KUKA KRL program: EPS_2_251497_STMH_A_20251003030554.src

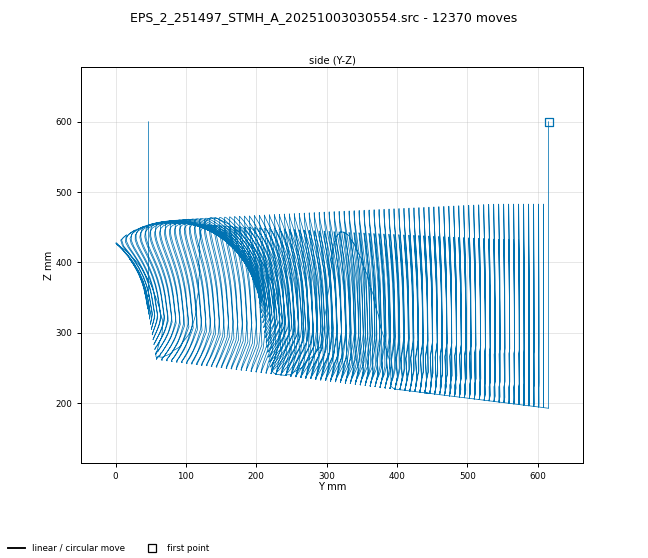
[picture p0: tool path of EPS_2_251497_STMH_A_20251003030554.src, 12370 of 12372 moves have a stored position in this frame; points joined in program order, loops and branches not executed]
&ACCESS RVP
&REL 4
&COMMENT QRS 19112012
&PARAM EDITMASK = *
DEF PART()
EXT BAS (BAS_COMMAND :IN,REAL :IN )
INT I
BAS (#INITMOV,0 )

;KUKA QRS Post kuka4.cps  Date:22-06-2017 !

File_ID=2874

QRS_PRE_INIT()

;Init var - Until changes are made in qrs_pre_init
Outlet_Square_prg=0
Inlet_1_Square_prg=0
Inlet_2_Square_prg=0
Inlet_3_Square_prg=0
Inlet_4_Square_prg=0
Inlet_5_Square_prg=0

Outlet_1={X 0.000, Y 540.910, Z 382.500, B 0.000, E1 0.000 }
Inlet_1={X 0.000, Y 544.470, Z 332.500, B 0.000, E1 230.000 }
Outlet_1_type=201
Inlet_1_type=201
;QRS#1=Sidecore dimensions
;QRS#2=200-8" PVC SDR 35
;QRS#3=200-8" PVC SDR 35
;QRS#4=
;QRS#5=
;QRS#6=
;QRS#7=
;QRS#8=
;QRS#9=12-08 PSX
;QRS#10=12-08 PSX
;QRS#11=
;QRS#12=
;QRS#13=
;QRS#14=
;QRS#15=
;QRS#16=1220x127x762 2,5'
;QRS#17=EPS Height
;QRS#18=483
;QRS#19=*
;QRS#20= UPDATED VERSION 22-06-2017
;QRS#21=*
Outlet_Square=0100
Inlet_1_Square=0100
Inlet_2_Square=0
Inlet_3_Square=0
Inlet_4_Square=0
Inlet_5_Square=0
Mill_Square=1
Outlet_Square_Prg=204
Inlet_1_Square_prg=204

QRS_INIT()

$ADVANCE=5

; T1
PTP {E1 173.565,E2 173.565}
PTP {X 0,Y 615.49,A -85,B 0,C 180,E1 173.565,E2 173.565,E3 0,E4 0,E5 0,E6 0}
QRS_SPEED_INIT()
LIN {X 0,Y 615.49,Z 600,A -85,B 0,C 180,E1 173.565,E2 173.565,E3 0,E4 0,E5 0,E6 0} C_VEL
LIN {X 0,Y 615.49,Z 202.871,A -85,B 0,C 180,E1 173.565,E2 173.565} C_VEL
LIN {X 0,Y 615.49,Z 194.7,A -85,B 0,C 180,E1 173.565,E2 173.565} C_VEL
LIN {X 0,Y 615.472,Z 192.7,A -85,B 0,C 180,E1 173.379,E2 173.379} C_VEL
LIN {X 0,Y 615.458,Z 192.696,A -85,B 0,C 180,E1 170.801,E2 170.801} C_VEL
LIN {X 0,Y 615.425,Z 192.697,A -85,B 0,C 180,E1 168.138,E2 168.138} C_VEL
LIN {X 0,Y 615.478,Z 192.701,A -85,B 0,C 180,E1 165.451,E2 165.451} C_VEL
LIN {X 0,Y 615.445,Z 192.694,A -85,B 0,C 180,E1 162.729,E2 162.729} C_VEL
LIN {X 0,Y 615.439,Z 192.695,A -85,B 0,C 180,E1 160.661,E2 160.661} C_VEL
LIN {X 0,Y 615.434,Z 192.695,A -85,B 0,C 180,E1 158.566,E2 158.566} C_VEL
LIN {X 0,Y 615.447,Z 192.698,A -85,B 0,C 180,E1 155.986,E2 155.986} C_VEL
LIN {X 0,Y 615.494,Z 192.701,A -85,B 0,C 180,E1 153.556,E2 153.556} C_VEL
LIN {X 0,Y 615.489,Z 192.693,A -85,B 0,C 180,E1 151.342,E2 151.342} C_VEL
LIN {X 0,Y 615.451,Z 192.692,A -85,B 0,C 180,E1 148.909,E2 148.909} C_VEL
LIN {X 0,Y 615.438,Z 192.695,A -85,B 0,C 180,E1 146.463,E2 146.463} C_VEL
LIN {X 0,Y 615.454,Z 192.697,A -85,B 0,C 180,E1 144.162,E2 144.162} C_VEL
LIN {X 0,Y 615.483,Z 192.699,A -85,B 0,C 180,E1 141.931,E2 141.931} C_VEL
LIN {X 0,Y 615.489,Z 192.688,A -85,B 0,C 180,E1 139.394,E2 139.394} C_VEL
LIN {X 0,Y 615.441,Z 192.694,A -85,B 0,C 180,E1 136.752,E2 136.752} C_VEL
LIN {X 0,Y 615.483,Z 192.702,A -85,B 0,C 180,E1 133.997,E2 133.997} C_VEL
LIN {X 0,Y 615.456,Z 192.69,A -85,B 0,C 180,E1 131.091,E2 131.091} C_VEL
LIN {X 0,Y 615.446,Z 192.692,A -85,B 0,C 180,E1 128.902,E2 128.902} C_VEL
LIN {X 0,Y 615.466,Z 192.697,A -85,B 0,C 180,E1 126.421,E2 126.421} C_VEL
LIN {X 0,Y 615.487,Z 192.686,A -85,B 0,C 180,E1 123.535,E2 123.535} C_VEL
LIN {X 0,Y 615.452,Z 192.692,A -85,B 0,C 180,E1 120.918,E2 120.918} C_VEL
LIN {X 0,Y 615.473,Z 192.699,A -85,B 0,C 180,E1 118.448,E2 118.448} C_VEL
LIN {X 0,Y 615.483,Z 192.685,A -85,B 0,C 180,E1 115.568,E2 115.568} C_VEL
LIN {X 0,Y 615.461,Z 192.694,A -85,B 0,C 180,E1 112.843,E2 112.843} C_VEL
LIN {X 0,Y 615.491,Z 192.69,A -85,B 0,C 180,E1 110.03,E2 110.03} C_VEL
LIN {X 0,Y 615.461,Z 192.689,A -85,B 0,C 180,E1 107.269,E2 107.269} C_VEL
LIN {X 0,Y 615.488,Z 192.702,A -85,B 0,C 180,E1 104.547,E2 104.547} C_VEL
LIN {X 0,Y 615.486,Z 192.685,A -85,B 0,C 180,E1 101.859,E2 101.859} C_VEL
LIN {X 0,Y 615.462,Z 192.692,A -85,B 0,C 180,E1 99.198,E2 99.198} C_VEL
LIN {X 0,Y 615.489,Z 192.698,A -85,B 0,C 180,E1 96.556,E2 96.556} C_VEL
LIN {X 0,Y 615.486,Z 192.684,A -85,B 0,C 180,E1 93.928,E2 93.928} C_VEL
LIN {X 0,Y 615.464,Z 192.692,A -85,B 0,C 180,E1 91.308,E2 91.308} C_VEL
LIN {X 0,Y 615.489,Z 192.698,A -85,B 0,C 180,E1 88.692,E2 88.692} C_VEL
LIN {X 0,Y 615.487,Z 192.683,A -85,B 0,C 180,E1 86.072,E2 86.072} C_VEL
LIN {X 0,Y 615.468,Z 192.692,A -85,B 0,C 180,E1 83.436,E2 83.436} C_VEL
LIN {X 0,Y 615.487,Z 192.697,A -85,B 0,C 180,E1 80.802,E2 80.802} C_VEL
LIN {X 0,Y 615.487,Z 192.683,A -85,B 0,C 180,E1 78.14,E2 78.14} C_VEL
LIN {X 0,Y 615.476,Z 192.693,A -85,B 0,C 180,E1 75.452,E2 75.452} C_VEL
LIN {X 0,Y 615.481,Z 192.692,A -85,B 0,C 180,E1 72.731,E2 72.731} C_VEL
LIN {X 0,Y 615.482,Z 192.685,A -85,B 0,C 180,E1 69.969,E2 69.969} C_VEL
LIN {X 0,Y 615.49,Z 192.7,A -85,B 0,C 180,E1 67.158,E2 67.158} C_VEL
LIN {X 0,Y 615.499,Z 192.68,A -85,B 0,C 180,E1 64.288,E2 64.288} C_VEL
LIN {X 0,Y 615.486,Z 192.703,A -85,B 0,C 180,E1 61.345,E2 61.345} C_VEL
LIN {X 0,Y 615.476,Z 192.691,A -85,B 0,C 180,E1 58.915,E2 58.915} C_VEL
LIN {X 0,Y 615.48,Z 192.89,A -85,B 0,C 180,E1 57.954,E2 57.954} C_VEL
LIN {X 0,Y 615.463,Z 208.033,A -85,B 0,C 180,E1 55.302,E2 55.302} C_VEL
LIN {X 0,Y 615.454,Z 222.372,A -85,B 0,C 180,E1 52.818,E2 52.818} C_VEL
LIN {X 0,Y 615.432,Z 329.039,A -85,B 0,C 180,E1 51.542,E2 51.542} C_VEL
LIN {X 0,Y 615.439,Z 342.064,A -85,B 0,C 180,E1 51.255,E2 51.255} C_VEL
LIN {X 0,Y 615.473,Z 354.262,A -85,B 0,C 180,E1 50.856,E2 50.856} C_VEL
LIN {X 0,Y 615.491,Z 365.958,A -85,B 0,C 180,E1 50.342,E2 50.342} C_VEL
LIN {X 0,Y 615.479,Z 377.926,A -85,B 0,C 180,E1 49.656,E2 49.656} C_VEL
LIN {X 0,Y 615.496,Z 388.354,A -85,B 0,C 180,E1 48.904,E2 48.904} C_VEL
LIN {X 0,Y 615.499,Z 397.717,A -85,B 0,C 180,E1 48.073,E2 48.073} C_VEL
LIN {X 0,Y 615.496,Z 406.315,A -85,B 0,C 180,E1 47.128,E2 47.128} C_VEL
LIN {X 0,Y 615.495,Z 413.248,A -85,B 0,C 180,E1 46.192,E2 46.192} C_VEL
LIN {X 0,Y 615.496,Z 419.897,A -85,B 0,C 180,E1 45.067,E2 45.067} C_VEL
LIN {X 0,Y 615.493,Z 424.69,A -85,B 0,C 180,E1 44.005,E2 44.005} C_VEL
LIN {X 0,Y 615.495,Z 427.941,A -85,B 0,C 180,E1 43.055,E2 43.055} C_VEL
LIN {X 0,Y 615.496,Z 430.296,A -85,B 0,C 180,E1 42.088,E2 42.088} C_VEL
LIN {X 0,Y 615.494,Z 431.771,A -85,B 0,C 180,E1 41.102,E2 41.102} C_VEL
LIN {X 0,Y 615.492,Z 432.346,A -85,B 0,C 180,E1 39.749,E2 39.749} C_VEL
LIN {X 0,Y 615.494,Z 431.883,A -85,B 0,C 180,E1 38.904,E2 38.904} C_VEL
LIN {X 0,Y 615.494,Z 430.657,A -85,B 0,C 180,E1 38.021,E2 38.021} C_VEL
LIN {X 0,Y 615.497,Z 428.187,A -85,B 0,C 180,E1 36.946,E2 36.946} C_VEL
LIN {X 0,Y 615.496,Z 424.457,A -85,B 0,C 180,E1 35.844,E2 35.844} C_VEL
LIN {X 0,Y 615.495,Z 419.188,A -85,B 0,C 180,E1 34.711,E2 34.711} C_VEL
LIN {X 0,Y 615.496,Z 412.08,A -85,B 0,C 180,E1 33.545,E2 33.545} C_VEL
LIN {X 0,Y 615.499,Z 405.237,A -85,B 0,C 180,E1 32.651,E2 32.651} C_VEL
LIN {X 0,Y 615.497,Z 397.831,A -85,B 0,C 180,E1 31.849,E2 31.849} C_VEL
LIN {X 0,Y 615.496,Z 388.386,A -85,B 0,C 180,E1 31.008,E2 31.008} C_VEL
LIN {X 0,Y 615.472,Z 377.947,A -85,B 0,C 180,E1 30.255,E2 30.255} C_VEL
LIN {X 0,Y 615.467,Z 366.665,A -85,B 0,C 180,E1 29.604,E2 29.604} C_VEL
LIN {X 0,Y 615.495,Z 354.87,A -85,B 0,C 180,E1 29.078,E2 29.078} C_VEL
LIN {X 0,Y 615.488,Z 342.102,A -85,B 0,C 180,E1 28.658,E2 28.658} C_VEL
LIN {X 0,Y 615.477,Z 330.305,A -85,B 0,C 180,E1 28.392,E2 28.392} C_VEL
LIN {X 0,Y 615.472,Z 295.985,A -85,B 0,C 180,E1 27.967,E2 27.967} C_VEL
LIN {X 0,Y 615.484,Z 222.337,A -85,B 0,C 180,E1 27.087,E2 27.087} C_VEL
LIN {X 0,Y 615.491,Z 206.092,A -85,B 0,C 180,E1 24.272,E2 24.272} C_VEL
LIN {X 0,Y 615.439,Z 192.697,A -85,B 0,C 180,E1 21.917,E2 21.917} C_VEL
LIN {X 0,Y 615.443,Z 192.698,A -85,B 0,C 180,E1 20.034,E2 20.034} C_VEL
LIN {X 0,Y 615.435,Z 192.697,A -85,B 0,C 180,E1 17.958,E2 17.958} C_VEL
LIN {X 0,Y 615.431,Z 192.697,A -85,B 0,C 180,E1 15.906,E2 15.906} C_VEL
LIN {X 0,Y 615.428,Z 192.697,A -85,B 0,C 180,E1 13.875,E2 13.875} C_VEL
LIN {X 0,Y 615.425,Z 192.697,A -85,B 0,C 180,E1 11.862,E2 11.862} C_VEL
LIN {X 0,Y 615.458,Z 192.695,A -85,B 0,C 180,E1 9.199,E2 9.199} C_VEL
LIN {X 0,Y 615.464,Z 192.7,A -85,B 0,C 180,E1 6.557,E2 6.557} C_VEL
LIN {X 0,Y 615.42,Z 192.698,A -85,B 0,C 180,E1 3.929,E2 3.929} C_VEL
LIN {X 0,Y 615.454,Z 192.697,A -85,B 0,C 180,E1 1.308,E2 1.308} C_VEL
LIN {X 0,Y 615.461,Z 192.7,A -85,B 0,C 180,E1 -1.309,E2 -1.309} C_VEL
LIN {X 0,Y 615.414,Z 192.699,A -85,B 0,C 180,E1 -3.929,E2 -3.929} C_VEL
LIN {X 0,Y 615.452,Z 192.699,A -85,B 0,C 180,E1 -6.604,E2 -6.604} C_VEL
LIN {X 0,Y 615.455,Z 192.7,A -85,B 0,C 180,E1 -9.2,E2 -9.2} C_VEL
LIN {X 0,Y 615.412,Z 192.7,A -85,B 0,C 180,E1 -11.863,E2 -11.863} C_VEL
LIN {X 0,Y 615.462,Z 192.7,A -85,B 0,C 180,E1 -14.55,E2 -14.55} C_VEL
LIN {X 0,Y 615.439,Z 192.698,A -85,B 0,C 180,E1 -17.272,E2 -17.272} C_VEL
LIN {X 0,Y 615.432,Z 192.698,A -85,B 0,C 180,E1 -19.34,E2 -19.34} C_VEL
LIN {X 0,Y 615.426,Z 192.698,A -85,B 0,C 180,E1 -21.434,E2 -21.434} C_VEL
LIN {X 0,Y 615.421,Z 192.698,A -85,B 0,C 180,E1 -23.559,E2 -23.559} C_VEL
LIN {X 0,Y 615.421,Z 192.698,A -85,B 0,C 180,E1 -25.719,E2 -25.719} C_VEL
LIN {X 0,Y 615.484,Z 192.701,A -85,B 0,C 180,E1 -28.461,E2 -28.461} C_VEL
LIN {X 0,Y 615.446,Z 192.695,A -85,B 0,C 180,E1 -31.09,E2 -31.09} C_VEL
LIN {X 0,Y 615.431,Z 192.696,A -85,B 0,C 180,E1 -33.24,E2 -33.24} C_VEL
LIN {X 0,Y 615.428,Z 192.697,A -85,B 0,C 180,E1 -35.62,E2 -35.62} C_VEL
LIN {X 0,Y 615.464,Z 192.699,A -85,B 0,C 180,E1 -38.071,E2 -38.071} C_VEL
LIN {X 0,Y 615.488,Z 192.692,A -85,B 0,C 180,E1 -40.607,E2 -40.607} C_VEL
LIN {X 0,Y 615.434,Z 192.695,A -85,B 0,C 180,E1 -43.25,E2 -43.25} C_VEL
LIN {X 0,Y 615.47,Z 192.7,A -85,B 0,C 180,E1 -46.005,E2 -46.005} C_VEL
LIN {X 0,Y 615.45,Z 192.692,A -85,B 0,C 180,E1 -48.91,E2 -48.91} C_VEL
LIN {X 0,Y 615.438,Z 192.694,A -85,B 0,C 180,E1 -51.097,E2 -51.097} C_VEL
LIN {X 0,Y 615.451,Z 192.697,A -85,B 0,C 180,E1 -53.577,E2 -53.577} C_VEL
LIN {X 0,Y 615.486,Z 192.688,A -85,B 0,C 180,E1 -56.467,E2 -56.467} C_VEL
LIN {X 0,Y 615.443,Z 192.693,A -85,B 0,C 180,E1 -59.082,E2 -59.082} C_VEL
LIN {X 0,Y 615.463,Z 192.697,A -85,B 0,C 180,E1 -61.554,E2 -61.554} C_VEL
LIN {X 0,Y 615.481,Z 192.687,A -85,B 0,C 180,E1 -64.433,E2 -64.433} C_VEL
LIN {X 0,Y 615.447,Z 192.693,A -85,B 0,C 180,E1 -67.046,E2 -67.046} C_VEL
LIN {X 0,Y 615.483,Z 210.777,A -85,B 0,C 180,E1 -69.445,E2 -69.445} C_VEL
LIN {X 0,Y 615.489,Z 232.032,A -85,B 0,C 180,E1 -72.217,E2 -72.217} C_VEL
LIN {X 0,Y 615.494,Z 253.252,A -85,B 0,C 180,E1 -74.945,E2 -74.945} C_VEL
LIN {X 0,Y 615.452,Z 270.312,A -85,B 0,C 180,E1 -77.114,E2 -77.114} C_VEL
LIN {X 0,Y 615.478,Z 378.901,A -85,B 0,C 180,E1 -78.412,E2 -78.412} C_VEL
LIN {X 0,Y 615.47,Z 391.391,A -85,B 0,C 180,E1 -78.683,E2 -78.683} C_VEL
LIN {X 0,Y 615.486,Z 404.642,A -85,B 0,C 180,E1 -79.114,E2 -79.114} C_VEL
LIN {X 0,Y 615.483,Z 416.499,A -85,B 0,C 180,E1 -79.64,E2 -79.64} C_VEL
LIN {X 0,Y 615.495,Z 428.01,A -85,B 0,C 180,E1 -80.305,E2 -80.305} C_VEL
LIN {X 0,Y 615.499,Z 438.353,A -85,B 0,C 180,E1 -81.051,E2 -81.051} C_VEL
LIN {X 0,Y 615.497,Z 446.821,A -85,B 0,C 180,E1 -81.795,E2 -81.795} C_VEL
LIN {X 0,Y 615.496,Z 455.971,A -85,B 0,C 180,E1 -82.785,E2 -82.785} C_VEL
LIN {X 0,Y 615.497,Z 463.319,A -85,B 0,C 180,E1 -83.773,E2 -83.773} C_VEL
LIN {X 0,Y 615.498,Z 469.207,A -85,B 0,C 180,E1 -84.759,E2 -84.759} C_VEL
LIN {X 0,Y 615.494,Z 473.853,A -85,B 0,C 180,E1 -85.744,E2 -85.744} C_VEL
LIN {X 0,Y 615.494,Z 477.4,A -85,B 0,C 180,E1 -86.727,E2 -86.727} C_VEL
LIN {X 0,Y 615.497,Z 479.233,A -85,B 0,C 180,E1 -87.382,E2 -87.382} C_VEL
LIN {X 0,Y 615.499,Z 480.608,A -85,B 0,C 180,E1 -88.037,E2 -88.037} C_VEL
LIN {X 0,Y 615.496,Z 482.173,A -85,B 0,C 180,E1 -89.346,E2 -89.346} C_VEL
LIN {X 0,Y 615.494,Z 482.389,A -85,B 0,C 180,E1 -90,E2 -90} C_VEL
LIN {X 0,Y 615.495,Z 481.58,A -85,B 0,C 180,E1 -91.308,E2 -91.308} C_VEL
LIN {X 0,Y 615.499,Z 480.608,A -85,B 0,C 180,E1 -91.963,E2 -91.963} C_VEL
LIN {X 0,Y 615.497,Z 479.234,A -85,B 0,C 180,E1 -92.617,E2 -92.617} C_VEL
LIN {X 0,Y 615.496,Z 476.351,A -85,B 0,C 180,E1 -93.6,E2 -93.6} C_VEL
LIN {X 0,Y 615.498,Z 472.444,A -85,B 0,C 180,E1 -94.584,E2 -94.584} C_VEL
LIN {X 0,Y 615.499,Z 467.409,A -85,B 0,C 180,E1 -95.569,E2 -95.569} C_VEL
LIN {X 0,Y 615.496,Z 460.87,A -85,B 0,C 180,E1 -96.583,E2 -96.583} C_VEL
LIN {X 0,Y 615.497,Z 453.141,A -85,B 0,C 180,E1 -97.544,E2 -97.544} C_VEL
LIN {X 0,Y 615.498,Z 445.056,A -85,B 0,C 180,E1 -98.37,E2 -98.37} C_VEL
LIN {X 0,Y 615.499,Z 435.182,A -85,B 0,C 180,E1 -99.198,E2 -99.198} C_VEL
LIN {X 0,Y 615.492,Z 424.001,A -85,B 0,C 180,E1 -99.944,E2 -99.944} C_VEL
LIN {X 0,Y 615.485,Z 413.049,A -85,B 0,C 180,E1 -100.526,E2 -100.526} C_VEL
LIN {X 0,Y 615.476,Z 400.523,A -85,B 0,C 180,E1 -101.039,E2 -101.039} C_VEL
LIN {X 0,Y 615.471,Z 388.127,A -85,B 0,C 180,E1 -101.401,E2 -101.401} C_VEL
LIN {X 0,Y 615.482,Z 374.566,A -85,B 0,C 180,E1 -101.651,E2 -101.651} C_VEL
LIN {X 0,Y 615.452,Z 270.313,A -85,B 0,C 180,E1 -102.886,E2 -102.886} C_VEL
LIN {X 0,Y 615.487,Z 249.274,A -85,B 0,C 180,E1 -105.563,E2 -105.563} C_VEL
LIN {X 0,Y 615.456,Z 227.017,A -85,B 0,C 180,E1 -108.434,E2 -108.434} C_VEL
LIN {X 0,Y 615.482,Z 206.801,A -85,B 0,C 180,E1 -111.079,E2 -111.079} C_VEL
LIN {X 0,Y 615.447,Z 192.693,A -85,B 0,C 180,E1 -112.977,E2 -112.977} C_VEL
LIN {X 0,Y 615.499,Z 192.686,A -85,B 0,C 180,E1 -115.712,E2 -115.712} C_VEL
LIN {X 0,Y 615.449,Z 192.695,A -85,B 0,C 180,E1 -118.656,E2 -118.656} C_VEL
LIN {X 0,Y 615.447,Z 192.692,A -85,B 0,C 180,E1 -121.079,E2 -121.079} C_VEL
LIN {X 0,Y 615.493,Z 192.701,A -85,B 0,C 180,E1 -124.017,E2 -124.017} C_VEL
LIN {X 0,Y 615.451,Z 192.697,A -85,B 0,C 180,E1 -126.422,E2 -126.422} C_VEL
LIN {X 0,Y 615.444,Z 192.693,A -85,B 0,C 180,E1 -129.057,E2 -129.057} C_VEL
LIN {X 0,Y 615.487,Z 192.69,A -85,B 0,C 180,E1 -131.468,E2 -131.468} C_VEL
LIN {X 0,Y 615.459,Z 192.698,A -85,B 0,C 180,E1 -134.146,E2 -134.146} C_VEL
LIN {X 0,Y 615.435,Z 192.695,A -85,B 0,C 180,E1 -136.75,E2 -136.75} C_VEL
LIN {X 0,Y 615.488,Z 192.692,A -85,B 0,C 180,E1 -139.393,E2 -139.393} C_VEL
LIN {X 0,Y 615.458,Z 192.699,A -85,B 0,C 180,E1 -141.983,E2 -141.983} C_VEL
LIN {X 0,Y 615.428,Z 192.697,A -85,B 0,C 180,E1 -144.38,E2 -144.38} C_VEL
LIN {X 0,Y 615.433,Z 192.696,A -85,B 0,C 180,E1 -146.76,E2 -146.76} C_VEL
LIN {X 0,Y 615.463,Z 192.694,A -85,B 0,C 180,E1 -149.079,E2 -149.079} C_VEL
LIN {X 0,Y 615.485,Z 192.701,A -85,B 0,C 180,E1 -151.538,E2 -151.538} C_VEL
LIN {X 0,Y 615.422,Z 192.698,A -85,B 0,C 180,E1 -154.281,E2 -154.281} C_VEL
LIN {X 0,Y 615.484,Z 192.696,A -85,B 0,C 180,E1 -157.155,E2 -157.155} C_VEL
LIN {X 0,Y 615.426,Z 192.699,A -85,B 0,C 180,E1 -159.965,E2 -159.965} C_VEL
LIN {X 0,Y 615.42,Z 192.699,A -85,B 0,C 180,E1 -162.041,E2 -162.041} C_VEL
LIN {X 0,Y 615.416,Z 192.699,A -85,B 0,C 180,E1 -164.093,E2 -164.093} C_VEL
LIN {X 0,Y 615.414,Z 192.699,A -85,B 0,C 180,E1 -166.124,E2 -166.124} C_VEL
LIN {X 0,Y 615.453,Z 192.699,A -85,B 0,C 180,E1 -168.806,E2 -168.806} C_VEL
LIN {X 0,Y 615.447,Z 192.7,A -85,B 0,C 180,E1 -171.463,E2 -171.463} C_VEL
LIN {X 0,Y 615.412,Z 192.7,A -85,B 0,C 180,E1 -174.1,E2 -174.1} C_VEL
LIN {X 0,Y 615.46,Z 192.7,A -85,B 0,C 180,E1 -176.727,E2 -176.727} C_VEL
LIN {X 0,Y 615.452,Z 192.698,A -85,B 0,C 180,E1 -179.345,E2 -179.345} C_VEL
LIN {X 0,Y 615.417,Z 192.699,A -85,B 0,C 180,E1 -181.963,E2 -181.963} C_VEL
LIN {X 0,Y 615.462,Z 192.7,A -85,B 0,C 180,E1 -184.585,E2 -184.585} C_VEL
LIN {X 0,Y 615.472,Z 192.7,A -85,B 0,C 180,E1 -186.621,E2 -186.621} C_VEL
LIN {X 0,Y 614.789,Z 192.842,A -85,B 0,C 180,E1 -187.167,E2 -187.167} C_VEL
LIN {X 0,Y 611.948,Z 193.253,A -85,B 0,C 180,E1 -188.053,E2 -188.053} C_VEL
LIN {X 0,Y 609.551,Z 193.564,A -85,B 0,C 180,E1 -188.766,E2 -188.766} C_VEL
LIN {X 0,Y 608.508,Z 193.683,A -85,B 0,C 180,E1 -189.315,E2 -189.315} C_VEL
LIN {X 0,Y 608.415,Z 193.693,A -85,B 0,C 180,E1 -189.501,E2 -189.501} C_VEL
LIN {X 0,Y 608.41,Z 193.694,A -85,B 0,C 180,E1 -192.001,E2 -192.001} C_VEL
LIN {X 0,Y 608.452,Z 193.697,A -85,B 0,C 180,E1 -194.721,E2 -194.721} C_VEL
LIN {X 0,Y 608.448,Z 193.695,A -85,B 0,C 180,E1 -196.784,E2 -196.784} C_VEL
LIN {X 0,Y 608.448,Z 193.693,A -85,B 0,C 180,E1 -198.87,E2 -198.87} C_VEL
LIN {X 0,Y 608.448,Z 193.691,A -85,B 0,C 180,E1 -200.982,E2 -200.982} C_VEL
LIN {X 0,Y 608.424,Z 193.692,A -85,B 0,C 180,E1 -203.125,E2 -203.125} C_VEL
LIN {X 0,Y 608.418,Z 193.693,A -85,B 0,C 180,E1 -205.724,E2 -205.724} C_VEL
LIN {X 0,Y 608.471,Z 193.691,A -85,B 0,C 180,E1 -208.631,E2 -208.631} C_VEL
LIN {X 0,Y 608.431,Z 193.69,A -85,B 0,C 180,E1 -211.318,E2 -211.318} C_VEL
LIN {X 0,Y 608.433,Z 193.692,A -85,B 0,C 180,E1 -213.739,E2 -213.739} C_VEL
LIN {X 0,Y 608.444,Z 193.697,A -85,B 0,C 180,E1 -216.092,E2 -216.092} C_VEL
LIN {X 0,Y 608.447,Z 193.692,A -85,B 0,C 180,E1 -218.589,E2 -218.589} C_VEL
LIN {X 0,Y 608.414,Z 193.692,A -85,B 0,C 180,E1 -221.18,E2 -221.18} C_VEL
LIN {X 0,Y 608.459,Z 193.693,A -85,B 0,C 180,E1 -223.87,E2 -223.87} C_VEL
LIN {X 0,Y 608.455,Z 193.688,A -85,B 0,C 180,E1 -226.692,E2 -226.692} C_VEL
LIN {X 0,Y 608.432,Z 193.69,A -85,B 0,C 180,E1 -228.827,E2 -228.827} C_VEL
LIN {X 0,Y 608.442,Z 193.691,A -85,B 0,C 180,E1 -231.415,E2 -231.415} C_VEL
LIN {X 0,Y 608.461,Z 193.696,A -85,B 0,C 180,E1 -233.952,E2 -233.952} C_VEL
LIN {X 0,Y 608.466,Z 193.689,A -85,B 0,C 180,E1 -236.334,E2 -236.334} C_VEL
LIN {X 0,Y 608.456,Z 193.687,A -85,B 0,C 180,E1 -238.731,E2 -238.731} C_VEL
LIN {X 0,Y 608.453,Z 193.692,A -85,B 0,C 180,E1 -241.383,E2 -241.383} C_VEL
LIN {X 0,Y 608.474,Z 193.687,A -85,B 0,C 180,E1 -244.278,E2 -244.278} C_VEL
LIN {X 0,Y 608.434,Z 193.69,A -85,B 0,C 180,E1 -246.878,E2 -246.878} C_VEL
LIN {X 0,Y 608.463,Z 193.694,A -85,B 0,C 180,E1 -249.728,E2 -249.728} C_VEL
LIN {X 0,Y 608.438,Z 193.689,A -85,B 0,C 180,E1 -252.525,E2 -252.525} C_VEL
LIN {X 0,Y 608.47,Z 193.692,A -85,B 0,C 180,E1 -255.281,E2 -255.281} C_VEL
LIN {X 0,Y 608.462,Z 193.688,A -85,B 0,C 180,E1 -258.002,E2 -258.002} C_VEL
LIN {X 0,Y 608.453,Z 193.688,A -85,B 0,C 180,E1 -260.695,E2 -260.695} C_VEL
LIN {X 0,Y 608.476,Z 193.695,A -85,B 0,C 180,E1 -263.368,E2 -263.368} C_VEL
LIN {X 0,Y 608.456,Z 193.688,A -85,B 0,C 180,E1 -266.027,E2 -266.027} C_VEL
LIN {X 0,Y 608.451,Z 193.69,A -85,B 0,C 180,E1 -268.676,E2 -268.676} C_VEL
LIN {X 0,Y 608.472,Z 193.693,A -85,B 0,C 180,E1 -271.324,E2 -271.324} C_VEL
LIN {X 0,Y 608.455,Z 193.687,A -85,B 0,C 180,E1 -273.974,E2 -273.974} C_VEL
LIN {X 0,Y 608.438,Z 193.693,A -85,B 0,C 180,E1 -276.632,E2 -276.632} C_VEL
LIN {X 0,Y 608.472,Z 193.691,A -85,B 0,C 180,E1 -279.305,E2 -279.305} C_VEL
LIN {X 0,Y 608.459,Z 193.687,A -85,B 0,C 180,E1 -281.999,E2 -281.999} C_VEL
LIN {X 0,Y 608.467,Z 193.693,A -85,B 0,C 180,E1 -284.719,E2 -284.719} C_VEL
LIN {X 0,Y 608.449,Z 193.69,A -85,B 0,C 180,E1 -287.475,E2 -287.475} C_VEL
LIN {X 0,Y 608.458,Z 193.689,A -85,B 0,C 180,E1 -290.272,E2 -290.272} C_VEL
LIN {X 0,Y 608.451,Z 193.692,A -85,B 0,C 180,E1 -293.121,E2 -293.121} C_VEL
LIN {X 0,Y 608.476,Z 193.684,A -85,B 0,C 180,E1 -295.722,E2 -295.722} C_VEL
LIN {X 0,Y 608.47,Z 193.696,A -85,B 0,C 180,E1 -298.62,E2 -298.62} C_VEL
LIN {X 0,Y 608.463,Z 193.687,A -85,B 0,C 180,E1 -301.313,E2 -301.313} C_VEL
LIN {X 0,Y 608.491,Z 193.868,A -85,B 0,C 180,E1 -301.991,E2 -301.991} C_VEL
LIN {X 0,Y 608.448,Z 209.134,A -85,B 0,C 180,E1 -304.686,E2 -304.686} C_VEL
LIN {X 0,Y 608.448,Z 222.747,A -85,B 0,C 180,E1 -307.047,E2 -307.047} C_VEL
LIN {X 0,Y 608.488,Z 329.338,A -85,B 0,C 180,E1 -308.328,E2 -308.328} C_VEL
LIN {X 0,Y 608.476,Z 342.925,A -85,B 0,C 180,E1 -308.635,E2 -308.635} C_VEL
LIN {X 0,Y 608.51,Z 355.443,A -85,B 0,C 180,E1 -309.058,E2 -309.058} C_VEL
LIN {X 0,Y 608.514,Z 367.155,A -85,B 0,C 180,E1 -309.592,E2 -309.592} C_VEL
LIN {X 0,Y 608.484,Z 379.103,A -85,B 0,C 180,E1 -310.295,E2 -310.295} C_VEL
LIN {X 0,Y 608.485,Z 389.451,A -85,B 0,C 180,E1 -311.059,E2 -311.059} C_VEL
LIN {X 0,Y 608.458,Z 398.323,A -85,B 0,C 180,E1 -311.863,E2 -311.863} C_VEL
LIN {X 0,Y 608.464,Z 406.644,A -85,B 0,C 180,E1 -312.784,E2 -312.784} C_VEL
LIN {X 0,Y 608.438,Z 414.554,A -85,B 0,C 180,E1 -313.866,E2 -313.866} C_VEL
LIN {X 0,Y 608.454,Z 420.979,A -85,B 0,C 180,E1 -314.996,E2 -314.996} C_VEL
LIN {X 0,Y 608.428,Z 425.886,A -85,B 0,C 180,E1 -316.127,E2 -316.127} C_VEL
LIN {X 0,Y 608.431,Z 428.854,A -85,B 0,C 180,E1 -317.039,E2 -317.039} C_VEL
LIN {X 0,Y 608.424,Z 430.986,A -85,B 0,C 180,E1 -317.936,E2 -317.936} C_VEL
LIN {X 0,Y 608.428,Z 432.302,A -85,B 0,C 180,E1 -318.821,E2 -318.821} C_VEL
LIN {X 0,Y 608.419,Z 432.924,A -85,B 0,C 180,E1 -319.694,E2 -319.694} C_VEL
LIN {X 0,Y 608.439,Z 432.789,A -85,B 0,C 180,E1 -320.698,E2 -320.698} C_VEL
LIN {X 0,Y 608.443,Z 431.66,A -85,B 0,C 180,E1 -321.755,E2 -321.755} C_VEL
LIN {X 0,Y 608.43,Z 428.769,A -85,B 0,C 180,E1 -323.084,E2 -323.084} C_VEL
LIN {X 0,Y 608.444,Z 424.431,A -85,B 0,C 180,E1 -324.337,E2 -324.337} C_VEL
LIN {X 0,Y 608.429,Z 418.692,A -85,B 0,C 180,E1 -325.528,E2 -325.528} C_VEL
LIN {X 0,Y 608.44,Z 412.517,A -85,B 0,C 180,E1 -326.527,E2 -326.527} C_VEL
LIN {X 0,Y 608.465,Z 405.33,A -85,B 0,C 180,E1 -327.467,E2 -327.467} C_VEL
LIN {X 0,Y 608.46,Z 396.625,A -85,B 0,C 180,E1 -328.392,E2 -328.392} C_VEL
LIN {X 0,Y 608.483,Z 386.513,A -85,B 0,C 180,E1 -329.264,E2 -329.264} C_VEL
LIN {X 0,Y 608.461,Z 375.642,A -85,B 0,C 180,E1 -330.019,E2 -330.019} C_VEL
LIN {X 0,Y 608.492,Z 365.084,A -85,B 0,C 180,E1 -330.603,E2 -330.603} C_VEL
LIN {X 0,Y 608.536,Z 353.361,A -85,B 0,C 180,E1 -331.11,E2 -331.11} C_VEL
LIN {X 0,Y 608.544,Z 340.12,A -85,B 0,C 180,E1 -331.531,E2 -331.531} C_VEL
LIN {X 0,Y 608.537,Z 327.961,A -85,B 0,C 180,E1 -331.785,E2 -331.785} C_VEL
LIN {X 0,Y 608.457,Z 222.623,A -85,B 0,C 180,E1 -333.05,E2 -333.05} C_VEL
LIN {X 0,Y 608.47,Z 206.674,A -85,B 0,C 180,E1 -335.835,E2 -335.835} C_VEL
LIN {X 0,Y 608.422,Z 193.693,A -85,B 0,C 180,E1 -338.151,E2 -338.151} C_VEL
LIN {X 0,Y 608.405,Z 193.693,A -85,B 0,C 180,E1 -340.428,E2 -340.428} C_VEL
LIN {X 0,Y 608.407,Z 193.693,A -85,B 0,C 180,E1 -342.522,E2 -342.522} C_VEL
LIN {X 0,Y 608.428,Z 193.691,A -85,B 0,C 180,E1 -344.593,E2 -344.593} C_VEL
LIN {X 0,Y 608.457,Z 193.698,A -85,B 0,C 180,E1 -347.323,E2 -347.323} C_VEL
LIN {X 0,Y 608.45,Z 193.697,A -85,B 0,C 180,E1 -349.35,E2 -349.35} C_VEL
LIN {X 0,Y 608.419,Z 193.692,A -85,B 0,C 180,E1 -352.033,E2 -352.033} C_VEL
LIN {X 0,Y 608.431,Z 193.693,A -85,B 0,C 180,E1 -354.698,E2 -354.698} C_VEL
LIN {X 0,Y 608.45,Z 193.694,A -85,B 0,C 180,E1 -357.352,E2 -357.352} C_VEL
LIN {X 0,Y 608.408,Z 193.693,A -85,B 0,C 180,E1 -360,E2 -360} C_VEL
LIN {X 0,Y 608.439,Z 193.693,A -85,B 0,C 180,E1 -362.648,E2 -362.648} C_VEL
LIN {X 0,Y 608.432,Z 193.695,A -85,B 0,C 180,E1 -365.302,E2 -365.302} C_VEL
LIN {X 0,Y 608.408,Z 193.693,A -85,B 0,C 180,E1 -367.968,E2 -367.968} C_VEL
LIN {X 0,Y 608.434,Z 193.696,A -85,B 0,C 180,E1 -370.651,E2 -370.651} C_VEL
LIN {X 0,Y 608.417,Z 193.694,A -85,B 0,C 180,E1 -373.358,E2 -373.358} C_VEL
LIN {X 0,Y 608.42,Z 193.693,A -85,B 0,C 180,E1 -375.407,E2 -375.407} C_VEL
LIN {X 0,Y 608.399,Z 193.695,A -85,B 0,C 180,E1 -377.478,E2 -377.478} C_VEL
LIN {X 0,Y 608.396,Z 193.695,A -85,B 0,C 180,E1 -379.573,E2 -379.573} C_VEL
LIN {X 0,Y 608.412,Z 193.692,A -85,B 0,C 180,E1 -381.694,E2 -381.694} C_VEL
LIN {X 0,Y 608.42,Z 193.702,A -85,B 0,C 180,E1 -384.573,E2 -384.573} C_VEL
LIN {X 0,Y 608.4,Z 193.694,A -85,B 0,C 180,E1 -387.521,E2 -387.521} C_VEL
LIN {X 0,Y 608.417,Z 193.694,A -85,B 0,C 180,E1 -389.974,E2 -389.974} C_VEL
LIN {X 0,Y 608.459,Z 193.696,A -85,B 0,C 180,E1 -392.532,E2 -392.532} C_VEL
LIN {X 0,Y 608.402,Z 193.694,A -85,B 0,C 180,E1 -395.281,E2 -395.281} C_VEL
LIN {X 0,Y 608.433,Z 193.692,A -85,B 0,C 180,E1 -397.749,E2 -397.749} C_VEL
LIN {X 0,Y 608.446,Z 193.698,A -85,B 0,C 180,E1 -400.336,E2 -400.336} C_VEL
LIN {X 0,Y 608.416,Z 193.693,A -85,B 0,C 180,E1 -402.963,E2 -402.963} C_VEL
LIN {X 0,Y 608.413,Z 193.692,A -85,B 0,C 180,E1 -405.206,E2 -405.206} C_VEL
LIN {X 0,Y 608.448,Z 193.695,A -85,B 0,C 180,E1 -407.943,E2 -407.943} C_VEL
LIN {X 0,Y 608.449,Z 193.69,A -85,B 0,C 180,E1 -410.705,E2 -410.705} C_VEL
LIN {X 0,Y 608.413,Z 193.692,A -85,B 0,C 180,E1 -413.087,E2 -413.087} C_VEL
LIN {X 0,Y 608.442,Z 193.692,A -85,B 0,C 180,E1 -415.533,E2 -415.533} C_VEL
LIN {X 0,Y 608.454,Z 193.697,A -85,B 0,C 180,E1 -417.909,E2 -417.909} C_VEL
LIN {X 0,Y 608.478,Z 193.69,A -85,B 0,C 180,E1 -420.225,E2 -420.225} C_VEL
LIN {X 0,Y 608.448,Z 193.688,A -85,B 0,C 180,E1 -422.799,E2 -422.799} C_VEL
LIN {X 0,Y 608.436,Z 193.694,A -85,B 0,C 180,E1 -425.431,E2 -425.431} C_VEL
LIN {X 0,Y 608.448,Z 193.84,A -85,B 0,C 180,E1 -426.924,E2 -426.924} C_VEL
LIN {X 0,Y 608.579,Z 209.461,A -85,B 0,C 180,E1 -429.025,E2 -429.025} C_VEL
LIN {X 0,Y 608.522,Z 230.732,A -85,B 0,C 180,E1 -431.832,E2 -431.832} C_VEL
LIN {X 0,Y 608.489,Z 252.003,A -85,B 0,C 180,E1 -434.596,E2 -434.596} C_VEL
LIN {X 0,Y 608.449,Z 270.533,A -85,B 0,C 180,E1 -436.974,E2 -436.974} C_VEL
LIN {X 0,Y 608.538,Z 379.015,A -85,B 0,C 180,E1 -438.278,E2 -438.278} C_VEL
LIN {X 0,Y 608.505,Z 392.261,A -85,B 0,C 180,E1 -438.573,E2 -438.573} C_VEL
LIN {X 0,Y 608.512,Z 404.651,A -85,B 0,C 180,E1 -438.983,E2 -438.983} C_VEL
LIN {X 0,Y 608.504,Z 416.656,A -85,B 0,C 180,E1 -439.52,E2 -439.52} C_VEL
LIN {X 0,Y 608.486,Z 428.213,A -85,B 0,C 180,E1 -440.192,E2 -440.192} C_VEL
LIN {X 0,Y 608.485,Z 438.606,A -85,B 0,C 180,E1 -440.947,E2 -440.947} C_VEL
LIN {X 0,Y 608.475,Z 447.121,A -85,B 0,C 180,E1 -441.7,E2 -441.7} C_VEL
LIN {X 0,Y 608.47,Z 454.967,A -85,B 0,C 180,E1 -442.535,E2 -442.535} C_VEL
LIN {X 0,Y 608.46,Z 462.289,A -85,B 0,C 180,E1 -443.485,E2 -443.485} C_VEL
LIN {X 0,Y 608.45,Z 467.869,A -85,B 0,C 180,E1 -444.366,E2 -444.366} C_VEL
LIN {X 0,Y 608.432,Z 472.952,A -85,B 0,C 180,E1 -445.363,E2 -445.363} C_VEL
LIN {X 0,Y 608.449,Z 476.897,A -85,B 0,C 180,E1 -446.358,E2 -446.358} C_VEL
LIN {X 0,Y 608.425,Z 479.81,A -85,B 0,C 180,E1 -447.352,E2 -447.352} C_VEL
LIN {X 0,Y 608.444,Z 481.202,A -85,B 0,C 180,E1 -448.014,E2 -448.014} C_VEL
LIN {X 0,Y 608.438,Z 482.783,A -85,B 0,C 180,E1 -449.338,E2 -449.338} C_VEL
LIN {X 0,Y 608.434,Z 483,A -85,B 0,C 180,E1 -450,E2 -450} C_VEL
LIN {X 0,Y 608.448,Z 482.184,A -85,B 0,C 180,E1 -451.324,E2 -451.324} C_VEL
LIN {X 0,Y 608.444,Z 481.202,A -85,B 0,C 180,E1 -451.986,E2 -451.986} C_VEL
LIN {X 0,Y 608.425,Z 479.81,A -85,B 0,C 180,E1 -452.648,E2 -452.648} C_VEL
LIN {X 0,Y 608.449,Z 476.898,A -85,B 0,C 180,E1 -453.642,E2 -453.642} C_VEL
LIN {X 0,Y 608.432,Z 472.952,A -85,B 0,C 180,E1 -454.637,E2 -454.637} C_VEL
LIN {X 0,Y 608.437,Z 466.881,A -85,B 0,C 180,E1 -455.8,E2 -455.8} C_VEL
LIN {X 0,Y 608.461,Z 460.241,A -85,B 0,C 180,E1 -456.798,E2 -456.798} C_VEL
LIN {X 0,Y 608.455,Z 451.997,A -85,B 0,C 180,E1 -457.799,E2 -457.799} C_VEL
LIN {X 0,Y 608.472,Z 443.548,A -85,B 0,C 180,E1 -458.635,E2 -458.635} C_VEL
LIN {X 0,Y 608.479,Z 433.106,A -85,B 0,C 180,E1 -459.472,E2 -459.472} C_VEL
LIN {X 0,Y 608.496,Z 422.776,A -85,B 0,C 180,E1 -460.143,E2 -460.143} C_VEL
LIN {X 0,Y 608.519,Z 411.292,A -85,B 0,C 180,E1 -460.739,E2 -460.739} C_VEL
LIN {X 0,Y 608.524,Z 398.926,A -85,B 0,C 180,E1 -461.224,E2 -461.224} C_VEL
LIN {X 0,Y 608.535,Z 385.498,A -85,B 0,C 180,E1 -461.596,E2 -461.596} C_VEL
LIN {X 0,Y 608.548,Z 373.19,A -85,B 0,C 180,E1 -461.806,E2 -461.806} C_VEL
LIN {X 0,Y 608.438,Z 270.451,A -85,B 0,C 180,E1 -463.037,E2 -463.037} C_VEL
LIN {X 0,Y 608.5,Z 249.345,A -85,B 0,C 180,E1 -465.747,E2 -465.747} C_VEL
LIN {X 0,Y 608.5,Z 228.27,A -85,B 0,C 180,E1 -468.491,E2 -468.491} C_VEL
LIN {X 0,Y 608.557,Z 208.132,A -85,B 0,C 180,E1 -471.153,E2 -471.153} C_VEL
LIN {X 0,Y 608.446,Z 193.758,A -85,B 0,C 180,E1 -473.088,E2 -473.088} C_VEL
LIN {X 0,Y 608.474,Z 193.688,A -85,B 0,C 180,E1 -475.721,E2 -475.721} C_VEL
LIN {X 0,Y 608.445,Z 193.691,A -85,B 0,C 180,E1 -478.615,E2 -478.615} C_VEL
LIN {X 0,Y 608.45,Z 193.691,A -85,B 0,C 180,E1 -480.542,E2 -480.542} C_VEL
LIN {X 0,Y 608.43,Z 193.69,A -85,B 0,C 180,E1 -482.877,E2 -482.877} C_VEL
LIN {X 0,Y 608.43,Z 193.691,A -85,B 0,C 180,E1 -485.274,E2 -485.274} C_VEL
LIN {X 0,Y 608.45,Z 193.693,A -85,B 0,C 180,E1 -488.238,E2 -488.238} C_VEL
LIN {X 0,Y 608.422,Z 193.695,A -85,B 0,C 180,E1 -490.325,E2 -490.325} C_VEL
LIN {X 0,Y 608.414,Z 193.692,A -85,B 0,C 180,E1 -492.957,E2 -492.957} C_VEL
LIN {X 0,Y 608.451,Z 193.698,A -85,B 0,C 180,E1 -495.73,E2 -495.73} C_VEL
LIN {X 0,Y 608.453,Z 193.694,A -85,B 0,C 180,E1 -497.938,E2 -497.938} C_VEL
LIN {X 0,Y 608.403,Z 193.694,A -85,B 0,C 180,E1 -500.702,E2 -500.702} C_VEL
LIN {X 0,Y 608.427,Z 193.693,A -85,B 0,C 180,E1 -503.083,E2 -503.083} C_VEL
LIN {X 0,Y 608.454,Z 193.697,A -85,B 0,C 180,E1 -505.529,E2 -505.529} C_VEL
LIN {X 0,Y 608.443,Z 193.693,A -85,B 0,C 180,E1 -507.904,E2 -507.904} C_VEL
LIN {X 0,Y 608.411,Z 193.693,A -85,B 0,C 180,E1 -510.217,E2 -510.217} C_VEL
LIN {X 0,Y 608.435,Z 193.691,A -85,B 0,C 180,E1 -512.788,E2 -512.788} C_VEL
LIN {X 0,Y 608.43,Z 193.694,A -85,B 0,C 180,E1 -515.843,E2 -515.843} C_VEL
LIN {X 0,Y 608.413,Z 193.692,A -85,B 0,C 180,E1 -518.306,E2 -518.306} C_VEL
LIN {X 0,Y 608.396,Z 193.695,A -85,B 0,C 180,E1 -520.427,E2 -520.427} C_VEL
LIN {X 0,Y 608.441,Z 193.699,A -85,B 0,C 180,E1 -523.215,E2 -523.215} C_VEL
LIN {X 0,Y 608.411,Z 193.693,A -85,B 0,C 180,E1 -525.979,E2 -525.979} C_VEL
LIN {X 0,Y 608.428,Z 193.693,A -85,B 0,C 180,E1 -528.675,E2 -528.675} C_VEL
LIN {X 0,Y 608.416,Z 193.698,A -85,B 0,C 180,E1 -531.363,E2 -531.363} C_VEL
LIN {X 0,Y 608.433,Z 193.695,A -85,B 0,C 180,E1 -533.367,E2 -533.367} C_VEL
LIN {X 0,Y 608.384,Z 193.696,A -85,B 0,C 180,E1 -536.025,E2 -536.025} C_VEL
LIN {X 0,Y 608.439,Z 193.695,A -85,B 0,C 180,E1 -538.676,E2 -538.676} C_VEL
LIN {X 0,Y 608.434,Z 193.694,A -85,B 0,C 180,E1 -541.324,E2 -541.324} C_VEL
LIN {X 0,Y 608.39,Z 193.695,A -85,B 0,C 180,E1 -543.974,E2 -543.974} C_VEL
LIN {X 0,Y 608.453,Z 193.696,A -85,B 0,C 180,E1 -546.666,E2 -546.666} C_VEL
LIN {X 0,Y 608.415,Z 193.693,A -85,B 0,C 180,E1 -549.501,E2 -549.501} C_VEL
LIN {X 0,Y 607.723,Z 193.78,A -85,B 0,C 180,E1 -550.054,E2 -550.054} C_VEL
LIN {X 0,Y 604.853,Z 194.142,A -85,B 0,C 180,E1 -550.951,E2 -550.951} C_VEL
LIN {X 0,Y 602.457,Z 194.438,A -85,B 0,C 180,E1 -551.673,E2 -551.673} C_VEL
LIN {X 0,Y 601.452,Z 194.563,A -85,B 0,C 180,E1 -552.23,E2 -552.23} C_VEL
LIN {X 0,Y 601.381,Z 194.572,A -85,B 0,C 180,E1 -552.418,E2 -552.418} C_VEL
LIN {X 0,Y 601.397,Z 194.572,A -85,B 0,C 180,E1 -554.897,E2 -554.897} C_VEL
LIN {X 0,Y 601.393,Z 194.571,A -85,B 0,C 180,E1 -556.987,E2 -556.987} C_VEL
LIN {X 0,Y 601.387,Z 194.57,A -85,B 0,C 180,E1 -559.1,E2 -559.1} C_VEL
LIN {X 0,Y 601.403,Z 194.566,A -85,B 0,C 180,E1 -561.239,E2 -561.239} C_VEL
LIN {X 0,Y 601.421,Z 194.568,A -85,B 0,C 180,E1 -564.142,E2 -564.142} C_VEL
LIN {X 0,Y 601.415,Z 194.565,A -85,B 0,C 180,E1 -567.113,E2 -567.113} C_VEL
LIN {X 0,Y 601.383,Z 194.568,A -85,B 0,C 180,E1 -569.395,E2 -569.395} C_VEL
LIN {X 0,Y 601.384,Z 194.57,A -85,B 0,C 180,E1 -571.728,E2 -571.728} C_VEL
LIN {X 0,Y 601.4,Z 194.574,A -85,B 0,C 180,E1 -574.12,E2 -574.12} C_VEL
LIN {X 0,Y 601.383,Z 194.573,A -85,B 0,C 180,E1 -576.584,E2 -576.584} C_VEL
LIN {X 0,Y 601.4,Z 194.566,A -85,B 0,C 180,E1 -579.127,E2 -579.127} C_VEL
LIN {X 0,Y 601.406,Z 194.57,A -85,B 0,C 180,E1 -581.766,E2 -581.766} C_VEL
LIN {X 0,Y 601.392,Z 194.57,A -85,B 0,C 180,E1 -584.539,E2 -584.539} C_VEL
LIN {X 0,Y 601.382,Z 194.569,A -85,B 0,C 180,E1 -587.333,E2 -587.333} C_VEL
LIN {X 0,Y 601.396,Z 194.577,A -85,B 0,C 180,E1 -590.009,E2 -590.009} C_VEL
LIN {X 0,Y 601.412,Z 194.565,A -85,B 0,C 180,E1 -592.621,E2 -592.621} C_VEL
LIN {X 0,Y 601.406,Z 194.566,A -85,B 0,C 180,E1 -595.072,E2 -595.072} C_VEL
LIN {X 0,Y 601.413,Z 194.569,A -85,B 0,C 180,E1 -597.487,E2 -597.487} C_VEL
LIN {X 0,Y 601.433,Z 194.571,A -85,B 0,C 180,E1 -599.85,E2 -599.85} C_VEL
LIN {X 0,Y 601.427,Z 194.563,A -85,B 0,C 180,E1 -602.891,E2 -602.891} C_VEL
LIN {X 0,Y 601.459,Z 194.566,A -85,B 0,C 180,E1 -605.863,E2 -605.863} C_VEL
LIN {X 0,Y 601.394,Z 194.567,A -85,B 0,C 180,E1 -608.763,E2 -608.763} C_VEL
LIN {X 0,Y 601.42,Z 194.573,A -85,B 0,C 180,E1 -611.61,E2 -611.61} C_VEL
LIN {X 0,Y 601.44,Z 194.568,A -85,B 0,C 180,E1 -613.715,E2 -613.715} C_VEL
LIN {X 0,Y 601.406,Z 194.565,A -85,B 0,C 180,E1 -616.485,E2 -616.485} C_VEL
LIN {X 0,Y 601.415,Z 194.571,A -85,B 0,C 180,E1 -619.225,E2 -619.225} C_VEL
LIN {X 0,Y 601.441,Z 194.563,A -85,B 0,C 180,E1 -621.94,E2 -621.94} C_VEL
LIN {X 0,Y 601.415,Z 194.565,A -85,B 0,C 180,E1 -624.636,E2 -624.636} C_VEL
LIN {X 0,Y 601.443,Z 194.57,A -85,B 0,C 180,E1 -627.321,E2 -627.321} C_VEL
LIN {X 0,Y 601.445,Z 194.561,A -85,B 0,C 180,E1 -630,E2 -630} C_VEL
LIN {X 0,Y 601.427,Z 194.566,A -85,B 0,C 180,E1 -632.679,E2 -632.679} C_VEL
LIN {X 0,Y 601.434,Z 194.568,A -85,B 0,C 180,E1 -635.363,E2 -635.363} C_VEL
LIN {X 0,Y 601.438,Z 194.561,A -85,B 0,C 180,E1 -638.06,E2 -638.06} C_VEL
LIN {X 0,Y 601.422,Z 194.574,A -85,B 0,C 180,E1 -641.012,E2 -641.012} C_VEL
LIN {X 0,Y 601.416,Z 194.566,A -85,B 0,C 180,E1 -643.514,E2 -643.514} C_VEL
LIN {X 0,Y 601.432,Z 194.564,A -85,B 0,C 180,E1 -646.285,E2 -646.285} C_VEL
LIN {X 0,Y 601.411,Z 194.571,A -85,B 0,C 180,E1 -649.097,E2 -649.097} C_VEL
LIN {X 0,Y 601.404,Z 194.569,A -85,B 0,C 180,E1 -651.237,E2 -651.237} C_VEL
LIN {X 0,Y 601.45,Z 194.561,A -85,B 0,C 180,E1 -654.138,E2 -654.138} C_VEL
LIN {X 0,Y 601.442,Z 194.565,A -85,B 0,C 180,E1 -657.108,E2 -657.108} C_VEL
LIN {X 0,Y 601.418,Z 194.565,A -85,B 0,C 180,E1 -659.39,E2 -659.39} C_VEL
LIN {X 0,Y 601.444,Z 194.673,A -85,B 0,C 180,E1 -661.918,E2 -661.918} C_VEL
LIN {X 0,Y 601.417,Z 209.236,A -85,B 0,C 180,E1 -664.52,E2 -664.52} C_VEL
LIN {X 0,Y 601.359,Z 222.612,A -85,B 0,C 180,E1 -666.882,E2 -666.882} C_VEL
LIN {X 0,Y 601.644,Z 229.528,A -85,B 0,C 180,E1 -666.979,E2 -666.979} C_VEL
LIN {X 0,Y 601.562,Z 329.06,A -85,B 0,C 180,E1 -668.186,E2 -668.186} C_VEL
LIN {X 0,Y 601.532,Z 342.272,A -85,B 0,C 180,E1 -668.483,E2 -668.483} C_VEL
LIN {X 0,Y 601.525,Z 355.19,A -85,B 0,C 180,E1 -668.919,E2 -668.919} C_VEL
LIN {X 0,Y 601.503,Z 366.764,A -85,B 0,C 180,E1 -669.448,E2 -669.448} C_VEL
LIN {X 0,Y 601.461,Z 377.775,A -85,B 0,C 180,E1 -670.092,E2 -670.092} C_VEL
LIN {X 0,Y 601.458,Z 388.366,A -85,B 0,C 180,E1 -670.865,E2 -670.865} C_VEL
LIN {X 0,Y 601.408,Z 398.276,A -85,B 0,C 180,E1 -671.761,E2 -671.761} C_VEL
LIN {X 0,Y 601.387,Z 406.396,A -85,B 0,C 180,E1 -672.667,E2 -672.667} C_VEL
LIN {X 0,Y 601.38,Z 413.17,A -85,B 0,C 180,E1 -673.585,E2 -673.585} C_VEL
LIN {X 0,Y 601.353,Z 420.073,A -85,B 0,C 180,E1 -674.753,E2 -674.753} C_VEL
LIN {X 0,Y 601.35,Z 425.38,A -85,B 0,C 180,E1 -675.943,E2 -675.943} C_VEL
LIN {X 0,Y 601.331,Z 428.524,A -85,B 0,C 180,E1 -676.879,E2 -676.879} C_VEL
LIN {X 0,Y 601.35,Z 429.914,A -85,B 0,C 180,E1 -677.409,E2 -677.409} C_VEL
LIN {X 0,Y 601.316,Z 431.818,A -85,B 0,C 180,E1 -678.411,E2 -678.411} C_VEL
LIN {X 0,Y 601.327,Z 432.821,A -85,B 0,C 180,E1 -679.429,E2 -679.429} C_VEL
LIN {X 0,Y 601.313,Z 432.907,A -85,B 0,C 180,E1 -680.471,E2 -680.471} C_VEL
LIN {X 0,Y 601.349,Z 431.738,A -85,B 0,C 180,E1 -681.727,E2 -681.727} C_VEL
LIN {X 0,Y 601.344,Z 429.035,A -85,B 0,C 180,E1 -683.019,E2 -683.019} C_VEL
LIN {X 0,Y 601.342,Z 425.027,A -85,B 0,C 180,E1 -684.243,E2 -684.243} C_VEL
LIN {X 0,Y 601.346,Z 419.353,A -85,B 0,C 180,E1 -685.471,E2 -685.471} C_VEL
LIN {X 0,Y 601.356,Z 413.021,A -85,B 0,C 180,E1 -686.528,E2 -686.528} C_VEL
LIN {X 0,Y 601.398,Z 405.918,A -85,B 0,C 180,E1 -687.483,E2 -687.483} C_VEL
LIN {X 0,Y 601.421,Z 397.23,A -85,B 0,C 180,E1 -688.433,E2 -688.433} C_VEL
LIN {X 0,Y 601.464,Z 386.759,A -85,B 0,C 180,E1 -689.353,E2 -689.353} C_VEL
LIN {X 0,Y 601.453,Z 375.781,A -85,B 0,C 180,E1 -690.128,E2 -690.128} C_VEL
LIN {X 0,Y 601.509,Z 364.131,A -85,B 0,C 180,E1 -690.773,E2 -690.773} C_VEL
LIN {X 0,Y 601.559,Z 351.288,A -85,B 0,C 180,E1 -691.319,E2 -691.319} C_VEL
LIN {X 0,Y 601.561,Z 338.233,A -85,B 0,C 180,E1 -691.713,E2 -691.713} C_VEL
LIN {X 0,Y 601.611,Z 324.944,A -85,B 0,C 180,E1 -691.965,E2 -691.965} C_VEL
LIN {X 0,Y 601.612,Z 223.962,A -85,B 0,C 180,E1 -693.179,E2 -693.179} C_VEL
LIN {X 0,Y 601.409,Z 222.564,A -85,B 0,C 180,E1 -693.216,E2 -693.216} C_VEL
LIN {X 0,Y 601.423,Z 206.58,A -85,B 0,C 180,E1 -696.042,E2 -696.042} C_VEL
LIN {X 0,Y 601.373,Z 194.572,A -85,B 0,C 180,E1 -698.197,E2 -698.197} C_VEL
LIN {X 0,Y 601.367,Z 194.571,A -85,B 0,C 180,E1 -700.19,E2 -700.19} C_VEL
LIN {X 0,Y 601.356,Z 194.572,A -85,B 0,C 180,E1 -702.311,E2 -702.311} C_VEL
LIN {X 0,Y 601.372,Z 194.57,A -85,B 0,C 180,E1 -704.408,E2 -704.408} C_VEL
LIN {X 0,Y 601.422,Z 194.572,A -85,B 0,C 180,E1 -707.172,E2 -707.172} C_VEL
LIN {X 0,Y 601.386,Z 194.57,A -85,B 0,C 180,E1 -709.904,E2 -709.904} C_VEL
LIN {X 0,Y 601.404,Z 194.567,A -85,B 0,C 180,E1 -712.615,E2 -712.615} C_VEL
LIN {X 0,Y 601.397,Z 194.575,A -85,B 0,C 180,E1 -715.308,E2 -715.308} C_VEL
LIN {X 0,Y 601.361,Z 194.571,A -85,B 0,C 180,E1 -717.991,E2 -717.991} C_VEL
LIN {X 0,Y 601.412,Z 194.569,A -85,B 0,C 180,E1 -720.67,E2 -720.67} C_VEL
LIN {X 0,Y 601.397,Z 194.571,A -85,B 0,C 180,E1 -723.35,E2 -723.35} C_VEL
LIN {X 0,Y 601.346,Z 194.573,A -85,B 0,C 180,E1 -726.038,E2 -726.038} C_VEL
LIN {X 0,Y 601.376,Z 194.569,A -85,B 0,C 180,E1 -728.062,E2 -728.062} C_VEL
LIN {X 0,Y 601.434,Z 194.569,A -85,B 0,C 180,E1 -731.048,E2 -731.048} C_VEL
LIN {X 0,Y 601.363,Z 194.571,A -85,B 0,C 180,E1 -734.094,E2 -734.094} C_VEL
LIN {X 0,Y 601.388,Z 194.574,A -85,B 0,C 180,E1 -736.987,E2 -736.987} C_VEL
LIN {X 0,Y 601.356,Z 194.572,A -85,B 0,C 180,E1 -739.811,E2 -739.811} C_VEL
LIN {X 0,Y 601.367,Z 194.571,A -85,B 0,C 180,E1 -741.961,E2 -741.961} C_VEL
LIN {X 0,Y 601.389,Z 194.572,A -85,B 0,C 180,E1 -744.297,E2 -744.297} C_VEL
LIN {X 0,Y 601.411,Z 194.567,A -85,B 0,C 180,E1 -747.113,E2 -747.113} C_VEL
LIN {X 0,Y 601.373,Z 194.569,A -85,B 0,C 180,E1 -749.396,E2 -749.396} C_VEL
LIN {X 0,Y 601.378,Z 194.57,A -85,B 0,C 180,E1 -751.729,E2 -751.729} C_VEL
LIN {X 0,Y 601.387,Z 194.573,A -85,B 0,C 180,E1 -754.121,E2 -754.121} C_VEL
LIN {X 0,Y 601.38,Z 194.575,A -85,B 0,C 180,E1 -756.585,E2 -756.585} C_VEL
LIN {X 0,Y 601.374,Z 194.57,A -85,B 0,C 180,E1 -759.13,E2 -759.13} C_VEL
LIN {X 0,Y 601.396,Z 194.569,A -85,B 0,C 180,E1 -761.768,E2 -761.768} C_VEL
LIN {X 0,Y 601.394,Z 194.572,A -85,B 0,C 180,E1 -764.539,E2 -764.539} C_VEL
LIN {X 0,Y 601.378,Z 194.569,A -85,B 0,C 180,E1 -767.333,E2 -767.333} C_VEL
LIN {X 0,Y 601.388,Z 194.576,A -85,B 0,C 180,E1 -770.008,E2 -770.008} C_VEL
LIN {X 0,Y 601.413,Z 194.567,A -85,B 0,C 180,E1 -772.621,E2 -772.621} C_VEL
LIN {X 0,Y 601.378,Z 194.569,A -85,B 0,C 180,E1 -775.07,E2 -775.07} C_VEL
LIN {X 0,Y 601.403,Z 194.569,A -85,B 0,C 180,E1 -777.487,E2 -777.487} C_VEL
LIN {X 0,Y 601.437,Z 194.571,A -85,B 0,C 180,E1 -779.851,E2 -779.851} C_VEL
LIN {X 0,Y 601.403,Z 194.566,A -85,B 0,C 180,E1 -782.89,E2 -782.89} C_VEL
LIN {X 0,Y 601.46,Z 194.569,A -85,B 0,C 180,E1 -785.863,E2 -785.863} C_VEL
LIN {X 0,Y 601.405,Z 194.67,A -85,B 0,C 180,E1 -786.751,E2 -786.751} C_VEL
LIN {X 0,Y 601.702,Z 199.692,A -85,B 0,C 180,E1 -787.449,E2 -787.449} C_VEL
LIN {X 0,Y 601.598,Z 220.096,A -85,B 0,C 180,E1 -790.199,E2 -790.199} C_VEL
LIN {X 0,Y 601.528,Z 241.368,A -85,B 0,C 180,E1 -793.019,E2 -793.019} C_VEL
LIN {X 0,Y 601.455,Z 262.639,A -85,B 0,C 180,E1 -795.797,E2 -795.797} C_VEL
LIN {X 0,Y 601.425,Z 270.533,A -85,B 0,C 180,E1 -796.819,E2 -796.819} C_VEL
LIN {X 0,Y 601.622,Z 285.569,A -85,B 0,C 180,E1 -797.006,E2 -797.006} C_VEL
LIN {X 0,Y 601.605,Z 379.015,A -85,B 0,C 180,E1 -798.141,E2 -798.141} C_VEL
LIN {X 0,Y 601.553,Z 392.261,A -85,B 0,C 180,E1 -798.439,E2 -798.439} C_VEL
LIN {X 0,Y 601.541,Z 404.659,A -85,B 0,C 180,E1 -798.854,E2 -798.854} C_VEL
LIN {X 0,Y 601.516,Z 416.654,A -85,B 0,C 180,E1 -799.397,E2 -799.397} C_VEL
LIN {X 0,Y 601.486,Z 428.215,A -85,B 0,C 180,E1 -800.077,E2 -800.077} C_VEL
LIN {X 0,Y 601.444,Z 438.607,A -85,B 0,C 180,E1 -800.84,E2 -800.84} C_VEL
LIN {X 0,Y 601.429,Z 447.121,A -85,B 0,C 180,E1 -801.602,E2 -801.602} C_VEL
LIN {X 0,Y 601.417,Z 454.967,A -85,B 0,C 180,E1 -802.447,E2 -802.447} C_VEL
LIN {X 0,Y 601.369,Z 462.228,A -85,B 0,C 180,E1 -803.399,E2 -803.399} C_VEL
LIN {X 0,Y 601.372,Z 467.869,A -85,B 0,C 180,E1 -804.3,E2 -804.3} C_VEL
LIN {X 0,Y 601.336,Z 472.952,A -85,B 0,C 180,E1 -805.308,E2 -805.308} C_VEL
LIN {X 0,Y 601.368,Z 476.897,A -85,B 0,C 180,E1 -806.315,E2 -806.315} C_VEL
LIN {X 0,Y 601.325,Z 479.81,A -85,B 0,C 180,E1 -807.321,E2 -807.321} C_VEL
LIN {X 0,Y 601.343,Z 481.202,A -85,B 0,C 180,E1 -807.991,E2 -807.991} C_VEL
LIN {X 0,Y 601.339,Z 482.784,A -85,B 0,C 180,E1 -809.33,E2 -809.33} C_VEL
LIN {X 0,Y 601.335,Z 483,A -85,B 0,C 180,E1 -810,E2 -810} C_VEL
LIN {X 0,Y 601.347,Z 482.185,A -85,B 0,C 180,E1 -811.339,E2 -811.339} C_VEL
LIN {X 0,Y 601.343,Z 481.202,A -85,B 0,C 180,E1 -812.009,E2 -812.009} C_VEL
LIN {X 0,Y 601.325,Z 479.81,A -85,B 0,C 180,E1 -812.679,E2 -812.679} C_VEL
LIN {X 0,Y 601.368,Z 476.898,A -85,B 0,C 180,E1 -813.685,E2 -813.685} C_VEL
LIN {X 0,Y 601.336,Z 472.952,A -85,B 0,C 180,E1 -814.692,E2 -814.692} C_VEL
LIN {X 0,Y 601.372,Z 466.881,A -85,B 0,C 180,E1 -815.868,E2 -815.868} C_VEL
LIN {X 0,Y 601.387,Z 460.242,A -85,B 0,C 180,E1 -816.879,E2 -816.879} C_VEL
LIN {X 0,Y 601.4,Z 451.998,A -85,B 0,C 180,E1 -817.891,E2 -817.891} C_VEL
LIN {X 0,Y 601.436,Z 443.548,A -85,B 0,C 180,E1 -818.737,E2 -818.737} C_VEL
LIN {X 0,Y 601.449,Z 433.108,A -85,B 0,C 180,E1 -819.584,E2 -819.584} C_VEL
LIN {X 0,Y 601.474,Z 422.778,A -85,B 0,C 180,E1 -820.263,E2 -820.263} C_VEL
LIN {X 0,Y 601.536,Z 410.617,A -85,B 0,C 180,E1 -820.895,E2 -820.895} C_VEL
LIN {X 0,Y 601.55,Z 398.256,A -85,B 0,C 180,E1 -821.378,E2 -821.378} C_VEL
LIN {X 0,Y 601.572,Z 385.497,A -85,B 0,C 180,E1 -821.732,E2 -821.732} C_VEL
LIN {X 0,Y 601.615,Z 373.19,A -85,B 0,C 180,E1 -821.945,E2 -821.945} C_VEL
LIN {X 0,Y 601.504,Z 271.271,A -85,B 0,C 180,E1 -823.168,E2 -823.168} C_VEL
LIN {X 0,Y 601.444,Z 270.284,A -85,B 0,C 180,E1 -823.213,E2 -823.213} C_VEL
LIN {X 0,Y 601.521,Z 248.016,A -85,B 0,C 180,E1 -826.108,E2 -826.108} C_VEL
LIN {X 0,Y 601.586,Z 225.415,A -85,B 0,C 180,E1 -829.091,E2 -829.091} C_VEL
LIN {X 0,Y 601.678,Z 204.144,A -85,B 0,C 180,E1 -831.946,E2 -831.946} C_VEL
LIN {X 0,Y 601.657,Z 196.167,A -85,B 0,C 180,E1 -833.034,E2 -833.034} C_VEL
LIN {X 0,Y 601.393,Z 194.571,A -85,B 0,C 180,E1 -833.272,E2 -833.272} C_VEL
LIN {X 0,Y 601.414,Z 194.57,A -85,B 0,C 180,E1 -835.867,E2 -835.867} C_VEL
LIN {X 0,Y 601.405,Z 194.567,A -85,B 0,C 180,E1 -838.783,E2 -838.783} C_VEL
LIN {X 0,Y 601.404,Z 194.567,A -85,B 0,C 180,E1 -841.452,E2 -841.452} C_VEL
LIN {X 0,Y 601.414,Z 194.573,A -85,B 0,C 180,E1 -844.115,E2 -844.115} C_VEL
LIN {X 0,Y 601.382,Z 194.57,A -85,B 0,C 180,E1 -846.58,E2 -846.58} C_VEL
LIN {X 0,Y 601.421,Z 194.568,A -85,B 0,C 180,E1 -849.533,E2 -849.533} C_VEL
LIN {X 0,Y 601.406,Z 194.574,A -85,B 0,C 180,E1 -851.761,E2 -851.761} C_VEL
LIN {X 0,Y 601.394,Z 194.568,A -85,B 0,C 180,E1 -854.532,E2 -854.532} C_VEL
LIN {X 0,Y 601.423,Z 194.568,A -85,B 0,C 180,E1 -857.401,E2 -857.401} C_VEL
LIN {X 0,Y 601.375,Z 194.57,A -85,B 0,C 180,E1 -860.464,E2 -860.464} C_VEL
LIN {X 0,Y 601.396,Z 194.566,A -85,B 0,C 180,E1 -862.614,E2 -862.614} C_VEL
LIN {X 0,Y 601.407,Z 194.567,A -85,B 0,C 180,E1 -865.067,E2 -865.067} C_VEL
LIN {X 0,Y 601.426,Z 194.572,A -85,B 0,C 180,E1 -867.484,E2 -867.484} C_VEL
LIN {X 0,Y 601.381,Z 194.573,A -85,B 0,C 180,E1 -869.848,E2 -869.848} C_VEL
LIN {X 0,Y 601.383,Z 194.569,A -85,B 0,C 180,E1 -872.13,E2 -872.13} C_VEL
LIN {X 0,Y 601.374,Z 194.569,A -85,B 0,C 180,E1 -874.38,E2 -874.38} C_VEL
LIN {X 0,Y 601.377,Z 194.569,A -85,B 0,C 180,E1 -876.588,E2 -876.588} C_VEL
LIN {X 0,Y 601.407,Z 194.573,A -85,B 0,C 180,E1 -879.477,E2 -879.477} C_VEL
LIN {X 0,Y 601.379,Z 194.574,A -85,B 0,C 180,E1 -881.607,E2 -881.607} C_VEL
LIN {X 0,Y 601.4,Z 194.569,A -85,B 0,C 180,E1 -883.712,E2 -883.712} C_VEL
LIN {X 0,Y 601.367,Z 194.571,A -85,B 0,C 180,E1 -886.483,E2 -886.483} C_VEL
LIN {X 0,Y 601.398,Z 194.575,A -85,B 0,C 180,E1 -889.223,E2 -889.223} C_VEL
LIN {X 0,Y 601.376,Z 194.569,A -85,B 0,C 180,E1 -891.938,E2 -891.938} C_VEL
LIN {X 0,Y 601.389,Z 194.571,A -85,B 0,C 180,E1 -894.635,E2 -894.635} C_VEL
LIN {X 0,Y 601.403,Z 194.57,A -85,B 0,C 180,E1 -897.321,E2 -897.321} C_VEL
LIN {X 0,Y 601.376,Z 194.569,A -85,B 0,C 180,E1 -900,E2 -900} C_VEL
LIN {X 0,Y 601.411,Z 194.572,A -85,B 0,C 180,E1 -902.679,E2 -902.679} C_VEL
LIN {X 0,Y 601.39,Z 194.57,A -85,B 0,C 180,E1 -905.364,E2 -905.364} C_VEL
LIN {X 0,Y 601.404,Z 194.567,A -85,B 0,C 180,E1 -907.385,E2 -907.385} C_VEL
LIN {X 0,Y 601.384,Z 194.569,A -85,B 0,C 180,E1 -910.096,E2 -910.096} C_VEL
LIN {X 0,Y 601.381,Z 194.572,A -85,B 0,C 180,E1 -912.418,E2 -912.418} C_VEL
LIN {X 0,Y 600.743,Z 194.656,A -85,B 0,C 180,E1 -912.978,E2 -912.978} C_VEL
LIN {X 0,Y 597.889,Z 195.011,A -85,B 0,C 180,E1 -913.885,E2 -913.885} C_VEL
LIN {X 0,Y 595.457,Z 195.316,A -85,B 0,C 180,E1 -914.615,E2 -914.615} C_VEL
LIN {X 0,Y 594.409,Z 195.44,A -85,B 0,C 180,E1 -915.179,E2 -915.179} C_VEL
LIN {X 0,Y 594.323,Z 195.448,A -85,B 0,C 180,E1 -915.37,E2 -915.37} C_VEL
LIN {X 0,Y 594.341,Z 195.446,A -85,B 0,C 180,E1 -917.905,E2 -917.905} C_VEL
LIN {X 0,Y 594.369,Z 195.446,A -85,B 0,C 180,E1 -920.931,E2 -920.931} C_VEL
LIN {X 0,Y 594.353,Z 195.444,A -85,B 0,C 180,E1 -923.705,E2 -923.705} C_VEL
LIN {X 0,Y 594.353,Z 195.449,A -85,B 0,C 180,E1 -926.701,E2 -926.701} C_VEL
LIN {X 0,Y 594.377,Z 195.442,A -85,B 0,C 180,E1 -928.998,E2 -928.998} C_VEL
LIN {X 0,Y 594.355,Z 195.445,A -85,B 0,C 180,E1 -931.649,E2 -931.649} C_VEL
LIN {X 0,Y 594.365,Z 195.447,A -85,B 0,C 180,E1 -934.581,E2 -934.581} C_VEL
LIN {X 0,Y 594.349,Z 195.444,A -85,B 0,C 180,E1 -937.089,E2 -937.089} C_VEL
LIN {X 0,Y 594.357,Z 195.447,A -85,B 0,C 180,E1 -939.78,E2 -939.78} C_VEL
LIN {X 0,Y 594.363,Z 195.449,A -85,B 0,C 180,E1 -942.376,E2 -942.376} C_VEL
LIN {X 0,Y 594.33,Z 195.447,A -85,B 0,C 180,E1 -945.194,E2 -945.194} C_VEL
LIN {X 0,Y 594.367,Z 195.45,A -85,B 0,C 180,E1 -948.153,E2 -948.153} C_VEL
LIN {X 0,Y 594.374,Z 195.446,A -85,B 0,C 180,E1 -950.325,E2 -950.325} C_VEL
LIN {X 0,Y 594.361,Z 195.443,A -85,B 0,C 180,E1 -952.916,E2 -952.916} C_VEL
LIN {X 0,Y 594.369,Z 195.453,A -85,B 0,C 180,E1 -955.863,E2 -955.863} C_VEL
LIN {X 0,Y 594.373,Z 195.442,A -85,B 0,C 180,E1 -958.654,E2 -958.654} C_VEL
LIN {X 0,Y 594.367,Z 195.443,A -85,B 0,C 180,E1 -961.045,E2 -961.045} C_VEL
LIN {X 0,Y 594.387,Z 195.445,A -85,B 0,C 180,E1 -963.977,E2 -963.977} C_VEL
LIN {X 0,Y 594.385,Z 195.441,A -85,B 0,C 180,E1 -966.299,E2 -966.299} C_VEL
LIN {X 0,Y 594.395,Z 195.443,A -85,B 0,C 180,E1 -969.227,E2 -969.227} C_VEL
LIN {X 0,Y 594.348,Z 195.447,A -85,B 0,C 180,E1 -972.097,E2 -972.097} C_VEL
LIN {X 0,Y 594.36,Z 195.444,A -85,B 0,C 180,E1 -974.221,E2 -974.221} C_VEL
LIN {X 0,Y 594.374,Z 195.441,A -85,B 0,C 180,E1 -976.322,E2 -976.322} C_VEL
LIN {X 0,Y 594.373,Z 195.446,A -85,B 0,C 180,E1 -979.096,E2 -979.096} C_VEL
LIN {X 0,Y 594.417,Z 195.439,A -85,B 0,C 180,E1 -981.844,E2 -981.844} C_VEL
LIN {X 0,Y 594.384,Z 195.441,A -85,B 0,C 180,E1 -984.573,E2 -984.573} C_VEL
LIN {X 0,Y 594.408,Z 195.447,A -85,B 0,C 180,E1 -987.29,E2 -987.29} C_VEL
LIN {X 0,Y 594.414,Z 195.437,A -85,B 0,C 180,E1 -990,E2 -990} C_VEL
LIN {X 0,Y 594.395,Z 195.442,A -85,B 0,C 180,E1 -992.711,E2 -992.711} C_VEL
LIN {X 0,Y 594.399,Z 195.443,A -85,B 0,C 180,E1 -995.427,E2 -995.427} C_VEL
LIN {X 0,Y 594.411,Z 195.437,A -85,B 0,C 180,E1 -998.156,E2 -998.156} C_VEL
LIN {X 0,Y 594.386,Z 195.449,A -85,B 0,C 180,E1 -1001.073,E2 -1001.073} C_VEL
LIN {X 0,Y 594.38,Z 195.441,A -85,B 0,C 180,E1 -1003.677,E2 -1003.677} C_VEL
LIN {X 0,Y 594.387,Z 195.447,A -85,B 0,C 180,E1 -1006.717,E2 -1006.717} C_VEL
LIN {X 0,Y 594.362,Z 195.445,A -85,B 0,C 180,E1 -1009.332,E2 -1009.332} C_VEL
LIN {X 0,Y 594.361,Z 195.444,A -85,B 0,C 180,E1 -1011.501,E2 -1011.501} C_VEL
LIN {X 0,Y 594.378,Z 195.446,A -85,B 0,C 180,E1 -1014.444,E2 -1014.444} C_VEL
LIN {X 0,Y 594.379,Z 195.451,A -85,B 0,C 180,E1 -1016.697,E2 -1016.697} C_VEL
LIN {X 0,Y 594.376,Z 195.446,A -85,B 0,C 180,E1 -1018.995,E2 -1018.995} C_VEL
LIN {X 0,Y 594.423,Z 195.578,A -85,B 0,C 180,E1 -1021.861,E2 -1021.861} C_VEL
LIN {X 0,Y 594.411,Z 209.216,A -85,B 0,C 180,E1 -1024.329,E2 -1024.329} C_VEL
LIN {X 0,Y 594.315,Z 222.601,A -85,B 0,C 180,E1 -1026.721,E2 -1026.721} C_VEL
LIN {X 0,Y 594.744,Z 225.956,A -85,B 0,C 180,E1 -1026.781,E2 -1026.781} C_VEL
LIN {X 0,Y 594.629,Z 329.399,A -85,B 0,C 180,E1 -1028.052,E2 -1028.052} C_VEL
LIN {X 0,Y 594.561,Z 342.773,A -85,B 0,C 180,E1 -1028.36,E2 -1028.36} C_VEL
LIN {X 0,Y 594.556,Z 355.199,A -85,B 0,C 180,E1 -1028.787,E2 -1028.787} C_VEL
LIN {X 0,Y 594.509,Z 367.017,A -85,B 0,C 180,E1 -1029.335,E2 -1029.335} C_VEL
LIN {X 0,Y 594.441,Z 378.738,A -85,B 0,C 180,E1 -1030.038,E2 -1030.038} C_VEL
LIN {X 0,Y 594.415,Z 389.234,A -85,B 0,C 180,E1 -1030.827,E2 -1030.827} C_VEL
LIN {X 0,Y 594.376,Z 398.182,A -85,B 0,C 180,E1 -1031.653,E2 -1031.653} C_VEL
LIN {X 0,Y 594.315,Z 406.651,A -85,B 0,C 180,E1 -1032.61,E2 -1032.61} C_VEL
LIN {X 0,Y 594.299,Z 413.553,A -85,B 0,C 180,E1 -1033.565,E2 -1033.565} C_VEL
LIN {X 0,Y 594.273,Z 419.178,A -85,B 0,C 180,E1 -1034.521,E2 -1034.521} C_VEL
LIN {X 0,Y 594.273,Z 423.692,A -85,B 0,C 180,E1 -1035.473,E2 -1035.473} C_VEL
LIN {X 0,Y 594.253,Z 428.07,A -85,B 0,C 180,E1 -1036.691,E2 -1036.691} C_VEL
LIN {X 0,Y 594.253,Z 430.419,A -85,B 0,C 180,E1 -1037.615,E2 -1037.615} C_VEL
LIN {X 0,Y 594.211,Z 431.992,A -85,B 0,C 180,E1 -1038.522,E2 -1038.522} C_VEL
LIN {X 0,Y 594.245,Z 432.822,A -85,B 0,C 180,E1 -1039.423,E2 -1039.423} C_VEL
LIN {X 0,Y 594.211,Z 432.946,A -85,B 0,C 180,E1 -1040.307,E2 -1040.307} C_VEL
LIN {X 0,Y 594.226,Z 432.291,A -85,B 0,C 180,E1 -1041.307,E2 -1041.307} C_VEL
LIN {X 0,Y 594.23,Z 430.57,A -85,B 0,C 180,E1 -1042.403,E2 -1042.403} C_VEL
LIN {X 0,Y 594.251,Z 426.981,A -85,B 0,C 180,E1 -1043.749,E2 -1043.749} C_VEL
LIN {X 0,Y 594.256,Z 421.788,A -85,B 0,C 180,E1 -1045.046,E2 -1045.046} C_VEL
LIN {X 0,Y 594.288,Z 415.408,A -85,B 0,C 180,E1 -1046.233,E2 -1046.233} C_VEL
LIN {X 0,Y 594.312,Z 408.314,A -85,B 0,C 180,E1 -1047.269,E2 -1047.269} C_VEL
LIN {X 0,Y 594.359,Z 399.658,A -85,B 0,C 180,E1 -1048.283,E2 -1048.283} C_VEL
LIN {X 0,Y 594.413,Z 390.604,A -85,B 0,C 180,E1 -1049.147,E2 -1049.147} C_VEL
LIN {X 0,Y 594.435,Z 380.115,A -85,B 0,C 180,E1 -1049.96,E2 -1049.96} C_VEL
LIN {X 0,Y 594.47,Z 368.814,A -85,B 0,C 180,E1 -1050.657,E2 -1050.657} C_VEL
LIN {X 0,Y 594.575,Z 356.387,A -85,B 0,C 180,E1 -1051.254,E2 -1051.254} C_VEL
LIN {X 0,Y 594.634,Z 343.693,A -85,B 0,C 180,E1 -1051.703,E2 -1051.703} C_VEL
LIN {X 0,Y 594.65,Z 330.909,A -85,B 0,C 180,E1 -1052.01,E2 -1052.01} C_VEL
LIN {X 0,Y 594.657,Z 303.993,A -85,B 0,C 180,E1 -1052.364,E2 -1052.364} C_VEL
LIN {X 0,Y 594.604,Z 224.101,A -85,B 0,C 180,E1 -1053.335,E2 -1053.335} C_VEL
LIN {X 0,Y 594.382,Z 222.458,A -85,B 0,C 180,E1 -1053.393,E2 -1053.393} C_VEL
LIN {X 0,Y 594.408,Z 207.267,A -85,B 0,C 180,E1 -1056.112,E2 -1056.112} C_VEL
LIN {X 0,Y 594.346,Z 195.501,A -85,B 0,C 180,E1 -1058.246,E2 -1058.246} C_VEL
LIN {X 0,Y 594.331,Z 195.448,A -85,B 0,C 180,E1 -1060.665,E2 -1060.665} C_VEL
LIN {X 0,Y 594.387,Z 195.449,A -85,B 0,C 180,E1 -1063.515,E2 -1063.515} C_VEL
LIN {X 0,Y 594.333,Z 195.447,A -85,B 0,C 180,E1 -1066.32,E2 -1066.32} C_VEL
LIN {X 0,Y 594.378,Z 195.449,A -85,B 0,C 180,E1 -1069.095,E2 -1069.095} C_VEL
LIN {X 0,Y 594.364,Z 195.444,A -85,B 0,C 180,E1 -1071.843,E2 -1071.843} C_VEL
LIN {X 0,Y 594.315,Z 195.45,A -85,B 0,C 180,E1 -1073.891,E2 -1073.891} C_VEL
LIN {X 0,Y 594.303,Z 195.451,A -85,B 0,C 180,E1 -1075.931,E2 -1075.931} C_VEL
LIN {X 0,Y 594.332,Z 195.447,A -85,B 0,C 180,E1 -1077.967,E2 -1077.967} C_VEL
LIN {X 0,Y 594.381,Z 195.445,A -85,B 0,C 180,E1 -1080.678,E2 -1080.678} C_VEL
LIN {X 0,Y 594.346,Z 195.449,A -85,B 0,C 180,E1 -1083.39,E2 -1083.39} C_VEL
LIN {X 0,Y 594.303,Z 195.45,A -85,B 0,C 180,E1 -1086.11,E2 -1086.11} C_VEL
LIN {X 0,Y 594.355,Z 195.444,A -85,B 0,C 180,E1 -1088.158,E2 -1088.158} C_VEL
LIN {X 0,Y 594.405,Z 195.443,A -85,B 0,C 180,E1 -1091.113,E2 -1091.113} C_VEL
LIN {X 0,Y 594.335,Z 195.45,A -85,B 0,C 180,E1 -1094.379,E2 -1094.379} C_VEL
LIN {X 0,Y 594.341,Z 195.448,A -85,B 0,C 180,E1 -1097.195,E2 -1097.195} C_VEL
LIN {X 0,Y 594.325,Z 195.449,A -85,B 0,C 180,E1 -1099.336,E2 -1099.336} C_VEL
LIN {X 0,Y 594.322,Z 195.448,A -85,B 0,C 180,E1 -1101.505,E2 -1101.505} C_VEL
LIN {X 0,Y 594.344,Z 195.445,A -85,B 0,C 180,E1 -1103.706,E2 -1103.706} C_VEL
LIN {X 0,Y 594.347,Z 195.453,A -85,B 0,C 180,E1 -1106.702,E2 -1106.702} C_VEL
LIN {X 0,Y 594.351,Z 195.447,A -85,B 0,C 180,E1 -1109,E2 -1109} C_VEL
LIN {X 0,Y 594.352,Z 195.444,A -85,B 0,C 180,E1 -1111.649,E2 -1111.649} C_VEL
LIN {X 0,Y 594.359,Z 195.45,A -85,B 0,C 180,E1 -1114.582,E2 -1114.582} C_VEL
LIN {X 0,Y 594.349,Z 195.445,A -85,B 0,C 180,E1 -1117.09,E2 -1117.09} C_VEL
LIN {X 0,Y 594.328,Z 195.449,A -85,B 0,C 180,E1 -1119.776,E2 -1119.776} C_VEL
LIN {X 0,Y 594.367,Z 195.45,A -85,B 0,C 180,E1 -1122.376,E2 -1122.376} C_VEL
LIN {X 0,Y 594.333,Z 195.446,A -85,B 0,C 180,E1 -1125.195,E2 -1125.195} C_VEL
LIN {X 0,Y 594.339,Z 195.448,A -85,B 0,C 180,E1 -1127.628,E2 -1127.628} C_VEL
LIN {X 0,Y 594.371,Z 195.448,A -85,B 0,C 180,E1 -1130.324,E2 -1130.324} C_VEL
LIN {X 0,Y 594.361,Z 195.443,A -85,B 0,C 180,E1 -1132.916,E2 -1132.916} C_VEL
LIN {X 0,Y 594.366,Z 195.451,A -85,B 0,C 180,E1 -1135.864,E2 -1135.864} C_VEL
LIN {X 0,Y 594.354,Z 195.445,A -85,B 0,C 180,E1 -1138.653,E2 -1138.653} C_VEL
LIN {X 0,Y 594.365,Z 195.443,A -85,B 0,C 180,E1 -1141.046,E2 -1141.046} C_VEL
LIN {X 0,Y 594.384,Z 195.449,A -85,B 0,C 180,E1 -1143.978,E2 -1143.978} C_VEL
LIN {X 0,Y 594.36,Z 195.501,A -85,B 0,C 180,E1 -1146.575,E2 -1146.575} C_VEL
LIN {X 0,Y 594.788,Z 199.662,A -85,B 0,C 180,E1 -1147.168,E2 -1147.168} C_VEL
LIN {X 0,Y 594.668,Z 220.096,A -85,B 0,C 180,E1 -1149.959,E2 -1149.959} C_VEL
LIN {X 0,Y 594.562,Z 240.038,A -85,B 0,C 180,E1 -1152.636,E2 -1152.636} C_VEL
LIN {X 0,Y 594.47,Z 261.31,A -85,B 0,C 180,E1 -1155.452,E2 -1155.452} C_VEL
LIN {X 0,Y 594.426,Z 270.533,A -85,B 0,C 180,E1 -1156.661,E2 -1156.661} C_VEL
LIN {X 0,Y 594.734,Z 276.627,A -85,B 0,C 180,E1 -1156.744,E2 -1156.744} C_VEL
LIN {X 0,Y 594.656,Z 379.015,A -85,B 0,C 180,E1 -1158,E2 -1158} C_VEL
LIN {X 0,Y 594.594,Z 392.262,A -85,B 0,C 180,E1 -1158.301,E2 -1158.301} C_VEL
LIN {X 0,Y 594.561,Z 405.237,A -85,B 0,C 180,E1 -1158.744,E2 -1158.744} C_VEL
LIN {X 0,Y 594.532,Z 416.653,A -85,B 0,C 180,E1 -1159.271,E2 -1159.271} C_VEL
LIN {X 0,Y 594.48,Z 428.217,A -85,B 0,C 180,E1 -1159.959,E2 -1159.959} C_VEL
LIN {X 0,Y 594.414,Z 438.609,A -85,B 0,C 180,E1 -1160.731,E2 -1160.731} C_VEL
LIN {X 0,Y 594.383,Z 447.121,A -85,B 0,C 180,E1 -1161.501,E2 -1161.501} C_VEL
LIN {X 0,Y 594.347,Z 454.967,A -85,B 0,C 180,E1 -1162.356,E2 -1162.356} C_VEL
LIN {X 0,Y 594.282,Z 462.816,A -85,B 0,C 180,E1 -1163.409,E2 -1163.409} C_VEL
LIN {X 0,Y 594.289,Z 469.683,A -85,B 0,C 180,E1 -1164.572,E2 -1164.572} C_VEL
LIN {X 0,Y 594.27,Z 474.373,A -85,B 0,C 180,E1 -1165.592,E2 -1165.592} C_VEL
LIN {X 0,Y 594.267,Z 477.957,A -85,B 0,C 180,E1 -1166.61,E2 -1166.61} C_VEL
LIN {X 0,Y 594.226,Z 479.809,A -85,B 0,C 180,E1 -1167.289,E2 -1167.289} C_VEL
LIN {X 0,Y 594.242,Z 481.201,A -85,B 0,C 180,E1 -1167.967,E2 -1167.967} C_VEL
LIN {X 0,Y 594.239,Z 482.784,A -85,B 0,C 180,E1 -1169.322,E2 -1169.322} C_VEL
LIN {X 0,Y 594.236,Z 483,A -85,B 0,C 180,E1 -1170,E2 -1170} C_VEL
LIN {X 0,Y 594.247,Z 482.185,A -85,B 0,C 180,E1 -1171.355,E2 -1171.355} C_VEL
LIN {X 0,Y 594.242,Z 481.202,A -85,B 0,C 180,E1 -1172.033,E2 -1172.033} C_VEL
LIN {X 0,Y 594.226,Z 479.81,A -85,B 0,C 180,E1 -1172.711,E2 -1172.711} C_VEL
LIN {X 0,Y 594.289,Z 476.898,A -85,B 0,C 180,E1 -1173.729,E2 -1173.729} C_VEL
LIN {X 0,Y 594.241,Z 472.952,A -85,B 0,C 180,E1 -1174.748,E2 -1174.748} C_VEL
LIN {X 0,Y 594.304,Z 466.882,A -85,B 0,C 180,E1 -1175.939,E2 -1175.939} C_VEL
LIN {X 0,Y 594.311,Z 460.242,A -85,B 0,C 180,E1 -1176.961,E2 -1176.961} C_VEL
LIN {X 0,Y 594.359,Z 451.998,A -85,B 0,C 180,E1 -1177.985,E2 -1177.985} C_VEL
LIN {X 0,Y 594.382,Z 443.549,A -85,B 0,C 180,E1 -1178.841,E2 -1178.841} C_VEL
LIN {X 0,Y 594.433,Z 433.11,A -85,B 0,C 180,E1 -1179.698,E2 -1179.698} C_VEL
LIN {X 0,Y 594.485,Z 422.779,A -85,B 0,C 180,E1 -1180.385,E2 -1180.385} C_VEL
LIN {X 0,Y 594.558,Z 411.726,A -85,B 0,C 180,E1 -1180.973,E2 -1180.973} C_VEL
LIN {X 0,Y 594.575,Z 399.744,A -85,B 0,C 180,E1 -1181.463,E2 -1181.463} C_VEL
LIN {X 0,Y 594.636,Z 386.409,A -85,B 0,C 180,E1 -1181.849,E2 -1181.849} C_VEL
LIN {X 0,Y 594.692,Z 373.19,A -85,B 0,C 180,E1 -1182.086,E2 -1182.086} C_VEL
LIN {X 0,Y 594.623,Z 272.053,A -85,B 0,C 180,E1 -1183.314,E2 -1183.314} C_VEL
LIN {X 0,Y 594.433,Z 270.451,A -85,B 0,C 180,E1 -1183.35,E2 -1183.35} C_VEL
LIN {X 0,Y 594.537,Z 248.016,A -85,B 0,C 180,E1 -1186.303,E2 -1186.303} C_VEL
LIN {X 0,Y 594.62,Z 227.106,A -85,B 0,C 180,E1 -1189.096,E2 -1189.096} C_VEL
LIN {X 0,Y 594.761,Z 206.803,A -85,B 0,C 180,E1 -1191.85,E2 -1191.85} C_VEL
LIN {X 0,Y 594.74,Z 197.496,A -85,B 0,C 180,E1 -1193.133,E2 -1193.133} C_VEL
LIN {X 0,Y 594.345,Z 195.451,A -85,B 0,C 180,E1 -1193.449,E2 -1193.449} C_VEL
LIN {X 0,Y 594.384,Z 195.449,A -85,B 0,C 180,E1 -1196.022,E2 -1196.022} C_VEL
LIN {X 0,Y 594.364,Z 195.443,A -85,B 0,C 180,E1 -1198.954,E2 -1198.954} C_VEL
LIN {X 0,Y 594.362,Z 195.447,A -85,B 0,C 180,E1 -1201.64,E2 -1201.64} C_VEL
LIN {X 0,Y 594.356,Z 195.445,A -85,B 0,C 180,E1 -1204.577,E2 -1204.577} C_VEL
LIN {X 0,Y 594.36,Z 195.443,A -85,B 0,C 180,E1 -1207.084,E2 -1207.084} C_VEL
LIN {X 0,Y 594.355,Z 195.452,A -85,B 0,C 180,E1 -1209.771,E2 -1209.771} C_VEL
LIN {X 0,Y 594.339,Z 195.448,A -85,B 0,C 180,E1 -1212.372,E2 -1212.372} C_VEL
LIN {X 0,Y 594.332,Z 195.448,A -85,B 0,C 180,E1 -1215.188,E2 -1215.188} C_VEL
LIN {X 0,Y 594.356,Z 195.447,A -85,B 0,C 180,E1 -1218.147,E2 -1218.147} C_VEL
LIN {X 0,Y 594.34,Z 195.447,A -85,B 0,C 180,E1 -1220.316,E2 -1220.316} C_VEL
LIN {X 0,Y 594.348,Z 195.445,A -85,B 0,C 180,E1 -1222.91,E2 -1222.91} C_VEL
LIN {X 0,Y 594.35,Z 195.45,A -85,B 0,C 180,E1 -1225.856,E2 -1225.856} C_VEL
LIN {X 0,Y 594.347,Z 195.445,A -85,B 0,C 180,E1 -1228.648,E2 -1228.648} C_VEL
LIN {X 0,Y 594.358,Z 195.449,A -85,B 0,C 180,E1 -1231.772,E2 -1231.772} C_VEL
LIN {X 0,Y 594.325,Z 195.449,A -85,B 0,C 180,E1 -1234.053,E2 -1234.053} C_VEL
LIN {X 0,Y 594.344,Z 195.445,A -85,B 0,C 180,E1 -1236.294,E2 -1236.294} C_VEL
LIN {X 0,Y 594.381,Z 195.449,A -85,B 0,C 180,E1 -1239.223,E2 -1239.223} C_VEL
LIN {X 0,Y 594.329,Z 195.447,A -85,B 0,C 180,E1 -1242.094,E2 -1242.094} C_VEL
LIN {X 0,Y 594.32,Z 195.448,A -85,B 0,C 180,E1 -1244.218,E2 -1244.218} C_VEL
LIN {X 0,Y 594.327,Z 195.455,A -85,B 0,C 180,E1 -1247.016,E2 -1247.016} C_VEL
LIN {X 0,Y 594.368,Z 195.452,A -85,B 0,C 180,E1 -1249.094,E2 -1249.094} C_VEL
LIN {X 0,Y 594.355,Z 195.444,A -85,B 0,C 180,E1 -1251.842,E2 -1251.842} C_VEL
LIN {X 0,Y 594.349,Z 195.447,A -85,B 0,C 180,E1 -1254.572,E2 -1254.572} C_VEL
LIN {X 0,Y 594.367,Z 195.447,A -85,B 0,C 180,E1 -1257.289,E2 -1257.289} C_VEL
LIN {X 0,Y 594.345,Z 195.445,A -85,B 0,C 180,E1 -1260,E2 -1260} C_VEL
LIN {X 0,Y 594.374,Z 195.449,A -85,B 0,C 180,E1 -1262.711,E2 -1262.711} C_VEL
LIN {X 0,Y 594.351,Z 195.446,A -85,B 0,C 180,E1 -1265.428,E2 -1265.428} C_VEL
LIN {X 0,Y 594.365,Z 195.443,A -85,B 0,C 180,E1 -1267.473,E2 -1267.473} C_VEL
LIN {X 0,Y 594.35,Z 195.447,A -85,B 0,C 180,E1 -1270.216,E2 -1270.216} C_VEL
LIN {X 0,Y 594.347,Z 195.448,A -85,B 0,C 180,E1 -1272.416,E2 -1272.416} C_VEL
LIN {X 0,Y 594.337,Z 195.449,A -85,B 0,C 180,E1 -1275.079,E2 -1275.079} C_VEL
LIN {X 0,Y 594.323,Z 195.448,A -85,B 0,C 180,E1 -1275.37,E2 -1275.37} C_VEL
LIN {X 0,Y 593.653,Z 195.533,A -85,B 0,C 180,E1 -1275.936,E2 -1275.936} C_VEL
LIN {X 0,Y 590.796,Z 195.893,A -85,B 0,C 180,E1 -1276.854,E2 -1276.854} C_VEL
LIN {X 0,Y 588.393,Z 196.191,A -85,B 0,C 180,E1 -1277.593,E2 -1277.593} C_VEL
LIN {X 0,Y 587.372,Z 196.317,A -85,B 0,C 180,E1 -1278.163,E2 -1278.163} C_VEL
LIN {X 0,Y 587.296,Z 196.326,A -85,B 0,C 180,E1 -1278.356,E2 -1278.356} C_VEL
LIN {X 0,Y 587.337,Z 196.32,A -85,B 0,C 180,E1 -1281.056,E2 -1281.056} C_VEL
LIN {X 0,Y 587.329,Z 196.319,A -85,B 0,C 180,E1 -1283.258,E2 -1283.258} C_VEL
LIN {X 0,Y 587.318,Z 196.328,A -85,B 0,C 180,E1 -1286.279,E2 -1286.279} C_VEL
LIN {X 0,Y 587.332,Z 196.319,A -85,B 0,C 180,E1 -1289.142,E2 -1289.142} C_VEL
LIN {X 0,Y 587.322,Z 196.323,A -85,B 0,C 180,E1 -1291.842,E2 -1291.842} C_VEL
LIN {X 0,Y 587.323,Z 196.329,A -85,B 0,C 180,E1 -1294.354,E2 -1294.354} C_VEL
LIN {X 0,Y 587.314,Z 196.323,A -85,B 0,C 180,E1 -1296.749,E2 -1296.749} C_VEL
LIN {X 0,Y 587.317,Z 196.321,A -85,B 0,C 180,E1 -1299.361,E2 -1299.361} C_VEL
LIN {X 0,Y 587.33,Z 196.329,A -85,B 0,C 180,E1 -1302.114,E2 -1302.114} C_VEL
LIN {X 0,Y 587.282,Z 196.325,A -85,B 0,C 180,E1 -1305.092,E2 -1305.092} C_VEL
LIN {X 0,Y 587.323,Z 196.329,A -85,B 0,C 180,E1 -1307.931,E2 -1307.931} C_VEL
LIN {X 0,Y 587.325,Z 196.32,A -85,B 0,C 180,E1 -1310.644,E2 -1310.644} C_VEL
LIN {X 0,Y 587.329,Z 196.32,A -85,B 0,C 180,E1 -1313.295,E2 -1313.295} C_VEL
LIN {X 0,Y 587.35,Z 196.325,A -85,B 0,C 180,E1 -1315.784,E2 -1315.784} C_VEL
LIN {X 0,Y 587.338,Z 196.321,A -85,B 0,C 180,E1 -1318.235,E2 -1318.235} C_VEL
LIN {X 0,Y 587.335,Z 196.318,A -85,B 0,C 180,E1 -1320.869,E2 -1320.869} C_VEL
LIN {X 0,Y 587.353,Z 196.324,A -85,B 0,C 180,E1 -1323.82,E2 -1323.82} C_VEL
LIN {X 0,Y 587.314,Z 196.321,A -85,B 0,C 180,E1 -1326.744,E2 -1326.744} C_VEL
LIN {X 0,Y 587.323,Z 196.328,A -85,B 0,C 180,E1 -1329.697,E2 -1329.697} C_VEL
LIN {X 0,Y 587.343,Z 196.317,A -85,B 0,C 180,E1 -1332.596,E2 -1332.596} C_VEL
LIN {X 0,Y 587.361,Z 196.321,A -85,B 0,C 180,E1 -1335.741,E2 -1335.741} C_VEL
LIN {X 0,Y 587.345,Z 196.319,A -85,B 0,C 180,E1 -1338.868,E2 -1338.868} C_VEL
LIN {X 0,Y 587.37,Z 196.318,A -85,B 0,C 180,E1 -1341.746,E2 -1341.746} C_VEL
LIN {X 0,Y 587.352,Z 196.316,A -85,B 0,C 180,E1 -1344.508,E2 -1344.508} C_VEL
LIN {X 0,Y 587.373,Z 196.324,A -85,B 0,C 180,E1 -1347.257,E2 -1347.257} C_VEL
LIN {X 0,Y 587.383,Z 196.313,A -85,B 0,C 180,E1 -1350,E2 -1350} C_VEL
LIN {X 0,Y 587.363,Z 196.318,A -85,B 0,C 180,E1 -1352.743,E2 -1352.743} C_VEL
LIN {X 0,Y 587.364,Z 196.318,A -85,B 0,C 180,E1 -1355.492,E2 -1355.492} C_VEL
LIN {X 0,Y 587.363,Z 196.315,A -85,B 0,C 180,E1 -1358.254,E2 -1358.254} C_VEL
LIN {X 0,Y 587.345,Z 196.325,A -85,B 0,C 180,E1 -1361.133,E2 -1361.133} C_VEL
LIN {X 0,Y 587.361,Z 196.316,A -85,B 0,C 180,E1 -1364.259,E2 -1364.259} C_VEL
LIN {X 0,Y 587.352,Z 196.318,A -85,B 0,C 180,E1 -1367.404,E2 -1367.404} C_VEL
LIN {X 0,Y 587.325,Z 196.322,A -85,B 0,C 180,E1 -1370.303,E2 -1370.303} C_VEL
LIN {X 0,Y 587.316,Z 196.323,A -85,B 0,C 180,E1 -1373.256,E2 -1373.256} C_VEL
LIN {X 0,Y 587.354,Z 196.319,A -85,B 0,C 180,E1 -1376.18,E2 -1376.18} C_VEL
LIN {X 0,Y 587.343,Z 196.321,A -85,B 0,C 180,E1 -1379.133,E2 -1379.133} C_VEL
LIN {X 0,Y 587.387,Z 196.51,A -85,B 0,C 180,E1 -1381.807,E2 -1381.807} C_VEL
LIN {X 0,Y 587.378,Z 210.406,A -85,B 0,C 180,E1 -1384.352,E2 -1384.352} C_VEL
LIN {X 0,Y 587.293,Z 222.607,A -85,B 0,C 180,E1 -1386.56,E2 -1386.56} C_VEL
LIN {X 0,Y 587.841,Z 227.4,A -85,B 0,C 180,E1 -1386.64,E2 -1386.64} C_VEL
LIN {X 0,Y 587.683,Z 329.439,A -85,B 0,C 180,E1 -1387.909,E2 -1387.909} C_VEL
LIN {X 0,Y 587.624,Z 342.421,A -85,B 0,C 180,E1 -1388.21,E2 -1388.21} C_VEL
LIN {X 0,Y 587.603,Z 354.896,A -85,B 0,C 180,E1 -1388.639,E2 -1388.639} C_VEL
LIN {X 0,Y 587.525,Z 367.468,A -85,B 0,C 180,E1 -1389.231,E2 -1389.231} C_VEL
LIN {X 0,Y 587.422,Z 379.538,A -85,B 0,C 180,E1 -1389.971,E2 -1389.971} C_VEL
LIN {X 0,Y 587.374,Z 390.1,A -85,B 0,C 180,E1 -1390.789,E2 -1390.789} C_VEL
LIN {X 0,Y 587.32,Z 399.82,A -85,B 0,C 180,E1 -1391.724,E2 -1391.724} C_VEL
LIN {X 0,Y 587.238,Z 408.609,A -85,B 0,C 180,E1 -1392.773,E2 -1392.773} C_VEL
LIN {X 0,Y 587.229,Z 415.083,A -85,B 0,C 180,E1 -1393.728,E2 -1393.728} C_VEL
LIN {X 0,Y 587.205,Z 421.471,A -85,B 0,C 180,E1 -1394.916,E2 -1394.916} C_VEL
LIN {X 0,Y 587.148,Z 426.066,A -85,B 0,C 180,E1 -1396.033,E2 -1396.033} C_VEL
LIN {X 0,Y 587.176,Z 428.992,A -85,B 0,C 180,E1 -1396.981,E2 -1396.981} C_VEL
LIN {X 0,Y 587.156,Z 431.078,A -85,B 0,C 180,E1 -1397.91,E2 -1397.91} C_VEL
LIN {X 0,Y 587.112,Z 432.488,A -85,B 0,C 180,E1 -1398.943,E2 -1398.943} C_VEL
LIN {X 0,Y 587.133,Z 432.995,A -85,B 0,C 180,E1 -1399.996,E2 -1399.996} C_VEL
LIN {X 0,Y 587.142,Z 432.551,A -85,B 0,C 180,E1 -1401.074,E2 -1401.074} C_VEL
LIN {X 0,Y 587.146,Z 430.683,A -85,B 0,C 180,E1 -1402.378,E2 -1402.378} C_VEL
LIN {X 0,Y 587.175,Z 427.266,A -85,B 0,C 180,E1 -1403.702,E2 -1403.702} C_VEL
LIN {X 0,Y 587.163,Z 422.584,A -85,B 0,C 180,E1 -1404.933,E2 -1404.933} C_VEL
LIN {X 0,Y 587.21,Z 416.139,A -85,B 0,C 180,E1 -1406.184,E2 -1406.184} C_VEL
LIN {X 0,Y 587.257,Z 409.795,A -85,B 0,C 180,E1 -1407.154,E2 -1407.154} C_VEL
LIN {X 0,Y 587.291,Z 401.092,A -85,B 0,C 180,E1 -1408.228,E2 -1408.228} C_VEL
LIN {X 0,Y 587.355,Z 391.692,A -85,B 0,C 180,E1 -1409.16,E2 -1409.16} C_VEL
LIN {X 0,Y 587.426,Z 380.755,A -85,B 0,C 180,E1 -1410.033,E2 -1410.033} C_VEL
LIN {X 0,Y 587.487,Z 370.306,A -85,B 0,C 180,E1 -1410.702,E2 -1410.702} C_VEL
LIN {X 0,Y 587.592,Z 357.791,A -85,B 0,C 180,E1 -1411.328,E2 -1411.328} C_VEL
LIN {X 0,Y 587.676,Z 344.753,A -85,B 0,C 180,E1 -1411.811,E2 -1411.811} C_VEL
LIN {X 0,Y 587.689,Z 332.267,A -85,B 0,C 180,E1 -1412.127,E2 -1412.127} C_VEL
LIN {X 0,Y 587.738,Z 313.399,A -85,B 0,C 180,E1 -1412.396,E2 -1412.396} C_VEL
LIN {X 0,Y 587.797,Z 225.595,A -85,B 0,C 180,E1 -1413.473,E2 -1413.473} C_VEL
LIN {X 0,Y 587.331,Z 222.608,A -85,B 0,C 180,E1 -1413.529,E2 -1413.529} C_VEL
LIN {X 0,Y 587.39,Z 207.956,A -85,B 0,C 180,E1 -1416.184,E2 -1416.184} C_VEL
LIN {X 0,Y 587.302,Z 196.337,A -85,B 0,C 180,E1 -1418.318,E2 -1418.318} C_VEL
LIN {X 0,Y 587.33,Z 196.325,A -85,B 0,C 180,E1 -1421.151,E2 -1421.151} C_VEL
LIN {X 0,Y 587.292,Z 196.326,A -85,B 0,C 180,E1 -1424.024,E2 -1424.024} C_VEL
LIN {X 0,Y 587.3,Z 196.326,A -85,B 0,C 180,E1 -1426.858,E2 -1426.858} C_VEL
LIN {X 0,Y 587.353,Z 196.322,A -85,B 0,C 180,E1 -1428.963,E2 -1428.963} C_VEL
LIN {X 0,Y 587.319,Z 196.323,A -85,B 0,C 180,E1 -1431.744,E2 -1431.744} C_VEL
LIN {X 0,Y 587.277,Z 196.327,A -85,B 0,C 180,E1 -1433.817,E2 -1433.817} C_VEL
LIN {X 0,Y 587.26,Z 196.329,A -85,B 0,C 180,E1 -1435.883,E2 -1435.883} C_VEL
LIN {X 0,Y 587.304,Z 196.323,A -85,B 0,C 180,E1 -1437.943,E2 -1437.943} C_VEL
LIN {X 0,Y 587.35,Z 196.321,A -85,B 0,C 180,E1 -1440.686,E2 -1440.686} C_VEL
LIN {X 0,Y 587.295,Z 196.327,A -85,B 0,C 180,E1 -1443.431,E2 -1443.431} C_VEL
LIN {X 0,Y 587.311,Z 196.323,A -85,B 0,C 180,E1 -1445.494,E2 -1445.494} C_VEL
LIN {X 0,Y 587.311,Z 196.322,A -85,B 0,C 180,E1 -1448.256,E2 -1448.256} C_VEL
LIN {X 0,Y 587.372,Z 196.318,A -85,B 0,C 180,E1 -1451.177,E2 -1451.177} C_VEL
LIN {X 0,Y 587.307,Z 196.324,A -85,B 0,C 180,E1 -1454.262,E2 -1454.262} C_VEL
LIN {X 0,Y 587.307,Z 196.323,A -85,B 0,C 180,E1 -1457.408,E2 -1457.408} C_VEL
LIN {X 0,Y 587.298,Z 196.323,A -85,B 0,C 180,E1 -1459.577,E2 -1459.577} C_VEL
LIN {X 0,Y 587.318,Z 196.329,A -85,B 0,C 180,E1 -1462.515,E2 -1462.515} C_VEL
LIN {X 0,Y 587.286,Z 196.324,A -85,B 0,C 180,E1 -1465.519,E2 -1465.519} C_VEL
LIN {X 0,Y 587.307,Z 196.323,A -85,B 0,C 180,E1 -1467.82,E2 -1467.82} C_VEL
LIN {X 0,Y 587.298,Z 196.333,A -85,B 0,C 180,E1 -1470.514,E2 -1470.514} C_VEL
LIN {X 0,Y 587.3,Z 196.324,A -85,B 0,C 180,E1 -1473.115,E2 -1473.115} C_VEL
LIN {X 0,Y 587.319,Z 196.323,A -85,B 0,C 180,E1 -1475.898,E2 -1475.898} C_VEL
LIN {X 0,Y 587.296,Z 196.331,A -85,B 0,C 180,E1 -1478.482,E2 -1478.482} C_VEL
LIN {X 0,Y 587.303,Z 196.322,A -85,B 0,C 180,E1 -1481.16,E2 -1481.16} C_VEL
LIN {X 0,Y 587.291,Z 196.329,A -85,B 0,C 180,E1 -1483.954,E2 -1483.954} C_VEL
LIN {X 0,Y 587.29,Z 196.324,A -85,B 0,C 180,E1 -1486.997,E2 -1486.997} C_VEL
LIN {X 0,Y 587.293,Z 196.328,A -85,B 0,C 180,E1 -1489.749,E2 -1489.749} C_VEL
LIN {X 0,Y 587.323,Z 196.325,A -85,B 0,C 180,E1 -1492.396,E2 -1492.396} C_VEL
LIN {X 0,Y 587.307,Z 196.322,A -85,B 0,C 180,E1 -1494.947,E2 -1494.947} C_VEL
LIN {X 0,Y 587.319,Z 196.323,A -85,B 0,C 180,E1 -1497.424,E2 -1497.424} C_VEL
LIN {X 0,Y 587.332,Z 196.328,A -85,B 0,C 180,E1 -1499.833,E2 -1499.833} C_VEL
LIN {X 0,Y 587.341,Z 196.322,A -85,B 0,C 180,E1 -1502.31,E2 -1502.31} C_VEL
LIN {X 0,Y 587.328,Z 196.321,A -85,B 0,C 180,E1 -1504.486,E2 -1504.486} C_VEL
LIN {X 0,Y 587.334,Z 196.366,A -85,B 0,C 180,E1 -1506.418,E2 -1506.418} C_VEL
LIN {X 0,Y 587.881,Z 200.506,A -85,B 0,C 180,E1 -1507.003,E2 -1507.003} C_VEL
LIN {X 0,Y 587.76,Z 220.096,A -85,B 0,C 180,E1 -1509.713,E2 -1509.713} C_VEL
LIN {X 0,Y 587.573,Z 241.368,A -85,B 0,C 180,E1 -1512.603,E2 -1512.603} C_VEL
LIN {X 0,Y 587.473,Z 261.31,A -85,B 0,C 180,E1 -1515.274,E2 -1515.274} C_VEL
LIN {X 0,Y 587.393,Z 270.533,A -85,B 0,C 180,E1 -1516.498,E2 -1516.498} C_VEL
LIN {X 0,Y 587.839,Z 274.838,A -85,B 0,C 180,E1 -1516.564,E2 -1516.564} C_VEL
LIN {X 0,Y 587.719,Z 379.015,A -85,B 0,C 180,E1 -1517.856,E2 -1517.856} C_VEL
LIN {X 0,Y 587.647,Z 392.263,A -85,B 0,C 180,E1 -1518.161,E2 -1518.161} C_VEL
LIN {X 0,Y 587.623,Z 404.624,A -85,B 0,C 180,E1 -1518.585,E2 -1518.585} C_VEL
LIN {X 0,Y 587.55,Z 416.651,A -85,B 0,C 180,E1 -1519.142,E2 -1519.142} C_VEL
LIN {X 0,Y 587.467,Z 428.218,A -85,B 0,C 180,E1 -1519.838,E2 -1519.838} C_VEL
LIN {X 0,Y 587.393,Z 438.611,A -85,B 0,C 180,E1 -1520.619,E2 -1520.619} C_VEL
LIN {X 0,Y 587.321,Z 447.122,A -85,B 0,C 180,E1 -1521.398,E2 -1521.398} C_VEL
LIN {X 0,Y 587.273,Z 454.967,A -85,B 0,C 180,E1 -1522.264,E2 -1522.264} C_VEL
LIN {X 0,Y 587.23,Z 461.474,A -85,B 0,C 180,E1 -1523.127,E2 -1523.127} C_VEL
LIN {X 0,Y 587.236,Z 467.87,A -85,B 0,C 180,E1 -1524.162,E2 -1524.162} C_VEL
LIN {X 0,Y 587.147,Z 472.952,A -85,B 0,C 180,E1 -1525.194,E2 -1525.194} C_VEL
LIN {X 0,Y 587.213,Z 476.897,A -85,B 0,C 180,E1 -1526.226,E2 -1526.226} C_VEL
LIN {X 0,Y 587.132,Z 479.809,A -85,B 0,C 180,E1 -1527.256,E2 -1527.256} C_VEL
LIN {X 0,Y 587.141,Z 481.2,A -85,B 0,C 180,E1 -1527.942,E2 -1527.942} C_VEL
LIN {X 0,Y 587.14,Z 482.784,A -85,B 0,C 180,E1 -1529.314,E2 -1529.314} C_VEL
LIN {X 0,Y 587.137,Z 483,A -85,B 0,C 180,E1 -1530,E2 -1530} C_VEL
LIN {X 0,Y 587.147,Z 482.186,A -85,B 0,C 180,E1 -1531.372,E2 -1531.372} C_VEL
LIN {X 0,Y 587.141,Z 481.201,A -85,B 0,C 180,E1 -1532.058,E2 -1532.058} C_VEL
LIN {X 0,Y 587.132,Z 479.811,A -85,B 0,C 180,E1 -1532.744,E2 -1532.744} C_VEL
LIN {X 0,Y 587.213,Z 476.897,A -85,B 0,C 180,E1 -1533.774,E2 -1533.774} C_VEL
LIN {X 0,Y 587.147,Z 472.952,A -85,B 0,C 180,E1 -1534.806,E2 -1534.806} C_VEL
LIN {X 0,Y 587.217,Z 466.881,A -85,B 0,C 180,E1 -1536.01,E2 -1536.01} C_VEL
LIN {X 0,Y 587.246,Z 460.243,A -85,B 0,C 180,E1 -1537.045,E2 -1537.045} C_VEL
LIN {X 0,Y 587.299,Z 451.998,A -85,B 0,C 180,E1 -1538.082,E2 -1538.082} C_VEL
LIN {X 0,Y 587.343,Z 443.549,A -85,B 0,C 180,E1 -1538.948,E2 -1538.948} C_VEL
LIN {X 0,Y 587.421,Z 433.112,A -85,B 0,C 180,E1 -1539.815,E2 -1539.815} C_VEL
LIN {X 0,Y 587.488,Z 422.777,A -85,B 0,C 180,E1 -1540.51,E2 -1540.51} C_VEL
LIN {X 0,Y 587.581,Z 410.841,A -85,B 0,C 180,E1 -1541.147,E2 -1541.147} C_VEL
LIN {X 0,Y 587.624,Z 398.637,A -85,B 0,C 180,E1 -1541.638,E2 -1541.638} C_VEL
LIN {X 0,Y 587.71,Z 385.494,A -85,B 0,C 180,E1 -1542.012,E2 -1542.012} C_VEL
LIN {X 0,Y 587.749,Z 373.19,A -85,B 0,C 180,E1 -1542.231,E2 -1542.231} C_VEL
LIN {X 0,Y 587.719,Z 272.612,A -85,B 0,C 180,E1 -1543.466,E2 -1543.466} C_VEL
LIN {X 0,Y 587.401,Z 270.451,A -85,B 0,C 180,E1 -1543.512,E2 -1543.512} C_VEL
LIN {X 0,Y 587.557,Z 249.345,A -85,B 0,C 180,E1 -1546.323,E2 -1546.323} C_VEL
LIN {X 0,Y 587.665,Z 227.459,A -85,B 0,C 180,E1 -1549.282,E2 -1549.282} C_VEL
LIN {X 0,Y 587.835,Z 209.462,A -85,B 0,C 180,E1 -1551.752,E2 -1551.752} C_VEL
LIN {X 0,Y 587.791,Z 198.81,A -85,B 0,C 180,E1 -1553.236,E2 -1553.236} C_VEL
LIN {X 0,Y 587.323,Z 196.327,A -85,B 0,C 180,E1 -1553.629,E2 -1553.629} C_VEL
LIN {X 0,Y 587.328,Z 196.328,A -85,B 0,C 180,E1 -1556.276,E2 -1556.276} C_VEL
LIN {X 0,Y 587.334,Z 196.319,A -85,B 0,C 180,E1 -1559.13,E2 -1559.13} C_VEL
LIN {X 0,Y 587.328,Z 196.326,A -85,B 0,C 180,E1 -1561.832,E2 -1561.832} C_VEL
LIN {X 0,Y 587.329,Z 196.323,A -85,B 0,C 180,E1 -1564.345,E2 -1564.345} C_VEL
LIN {X 0,Y 587.331,Z 196.319,A -85,B 0,C 180,E1 -1566.743,E2 -1566.743} C_VEL
LIN {X 0,Y 587.323,Z 196.322,A -85,B 0,C 180,E1 -1569.356,E2 -1569.356} C_VEL
LIN {X 0,Y 587.308,Z 196.327,A -85,B 0,C 180,E1 -1572.104,E2 -1572.104} C_VEL
LIN {X 0,Y 587.285,Z 196.324,A -85,B 0,C 180,E1 -1574.908,E2 -1574.908} C_VEL
LIN {X 0,Y 587.319,Z 196.327,A -85,B 0,C 180,E1 -1577.924,E2 -1577.924} C_VEL
LIN {X 0,Y 587.289,Z 196.325,A -85,B 0,C 180,E1 -1581.056,E2 -1581.056} C_VEL
LIN {X 0,Y 587.316,Z 196.325,A -85,B 0,C 180,E1 -1583.288,E2 -1583.288} C_VEL
LIN {X 0,Y 587.332,Z 196.325,A -85,B 0,C 180,E1 -1585.778,E2 -1585.778} C_VEL
LIN {X 0,Y 587.317,Z 196.321,A -85,B 0,C 180,E1 -1588.229,E2 -1588.229} C_VEL
LIN {X 0,Y 587.314,Z 196.322,A -85,B 0,C 180,E1 -1590.861,E2 -1590.861} C_VEL
LIN {X 0,Y 587.311,Z 196.325,A -85,B 0,C 180,E1 -1593.816,E2 -1593.816} C_VEL
LIN {X 0,Y 587.317,Z 196.322,A -85,B 0,C 180,E1 -1596.741,E2 -1596.741} C_VEL
LIN {X 0,Y 587.295,Z 196.327,A -85,B 0,C 180,E1 -1599.694,E2 -1599.694} C_VEL
LIN {X 0,Y 587.282,Z 196.326,A -85,B 0,C 180,E1 -1601.872,E2 -1601.872} C_VEL
LIN {X 0,Y 587.282,Z 196.325,A -85,B 0,C 180,E1 -1604.023,E2 -1604.023} C_VEL
LIN {X 0,Y 587.275,Z 196.33,A -85,B 0,C 180,E1 -1606.857,E2 -1606.857} C_VEL
LIN {X 0,Y 587.353,Z 196.323,A -85,B 0,C 180,E1 -1608.962,E2 -1608.962} C_VEL
LIN {X 0,Y 587.311,Z 196.322,A -85,B 0,C 180,E1 -1611.744,E2 -1611.744} C_VEL
LIN {X 0,Y 587.311,Z 196.323,A -85,B 0,C 180,E1 -1614.506,E2 -1614.506} C_VEL
LIN {X 0,Y 587.331,Z 196.324,A -85,B 0,C 180,E1 -1617.256,E2 -1617.256} C_VEL
LIN {X 0,Y 587.315,Z 196.321,A -85,B 0,C 180,E1 -1620,E2 -1620} C_VEL
LIN {X 0,Y 587.338,Z 196.326,A -85,B 0,C 180,E1 -1622.743,E2 -1622.743} C_VEL
LIN {X 0,Y 587.314,Z 196.322,A -85,B 0,C 180,E1 -1625.493,E2 -1625.493} C_VEL
LIN {X 0,Y 587.328,Z 196.32,A -85,B 0,C 180,E1 -1627.563,E2 -1627.563} C_VEL
LIN {X 0,Y 587.306,Z 196.326,A -85,B 0,C 180,E1 -1630.34,E2 -1630.34} C_VEL
LIN {X 0,Y 587.304,Z 196.328,A -85,B 0,C 180,E1 -1632.439,E2 -1632.439} C_VEL
LIN {X 0,Y 587.292,Z 196.325,A -85,B 0,C 180,E1 -1635.264,E2 -1635.264} C_VEL
LIN {X 0,Y 587.313,Z 196.321,A -85,B 0,C 180,E1 -1637.407,E2 -1637.407} C_VEL
LIN {X 0,Y 587.296,Z 196.326,A -85,B 0,C 180,E1 -1638.356,E2 -1638.356} C_VEL
LIN {X 0,Y 586.649,Z 196.409,A -85,B 0,C 180,E1 -1638.928,E2 -1638.928} C_VEL
LIN {X 0,Y 583.815,Z 196.76,A -85,B 0,C 180,E1 -1639.857,E2 -1639.857} C_VEL
LIN {X 0,Y 581.404,Z 197.066,A -85,B 0,C 180,E1 -1640.604,E2 -1640.604} C_VEL
LIN {X 0,Y 580.36,Z 197.189,A -85,B 0,C 180,E1 -1641.18,E2 -1641.18} C_VEL
LIN {X 0,Y 580.272,Z 197.198,A -85,B 0,C 180,E1 -1641.375,E2 -1641.375} C_VEL
LIN {X 0,Y 580.26,Z 197.2,A -85,B 0,C 180,E1 -1643.559,E2 -1643.559} C_VEL
LIN {X 0,Y 580.282,Z 197.206,A -85,B 0,C 180,E1 -1646.345,E2 -1646.345} C_VEL
LIN {X 0,Y 580.278,Z 197.197,A -85,B 0,C 180,E1 -1649.317,E2 -1649.317} C_VEL
LIN {X 0,Y 580.268,Z 197.207,A -85,B 0,C 180,E1 -1652.202,E2 -1652.202} C_VEL
LIN {X 0,Y 580.264,Z 197.202,A -85,B 0,C 180,E1 -1654.698,E2 -1654.698} C_VEL
LIN {X 0,Y 580.263,Z 197.199,A -85,B 0,C 180,E1 -1657.271,E2 -1657.271} C_VEL
LIN {X 0,Y 580.298,Z 197.203,A -85,B 0,C 180,E1 -1660.279,E2 -1660.279} C_VEL
LIN {X 0,Y 580.265,Z 197.201,A -85,B 0,C 180,E1 -1662.707,E2 -1662.707} C_VEL
LIN {X 0,Y 580.242,Z 197.205,A -85,B 0,C 180,E1 -1665.612,E2 -1665.612} C_VEL
LIN {X 0,Y 580.277,Z 197.198,A -85,B 0,C 180,E1 -1668.669,E2 -1668.669} C_VEL
LIN {X 0,Y 580.266,Z 197.199,A -85,B 0,C 180,E1 -1670.969,E2 -1670.969} C_VEL
LIN {X 0,Y 580.273,Z 197.203,A -85,B 0,C 180,E1 -1673.602,E2 -1673.602} C_VEL
LIN {X 0,Y 580.303,Z 197.199,A -85,B 0,C 180,E1 -1676.149,E2 -1676.149} C_VEL
LIN {X 0,Y 580.273,Z 197.198,A -85,B 0,C 180,E1 -1678.618,E2 -1678.618} C_VEL
LIN {X 0,Y 580.278,Z 197.198,A -85,B 0,C 180,E1 -1681.027,E2 -1681.027} C_VEL
LIN {X 0,Y 580.317,Z 197.202,A -85,B 0,C 180,E1 -1683.661,E2 -1683.661} C_VEL
LIN {X 0,Y 580.271,Z 197.199,A -85,B 0,C 180,E1 -1686.445,E2 -1686.445} C_VEL
LIN {X 0,Y 580.267,Z 197.206,A -85,B 0,C 180,E1 -1689.439,E2 -1689.439} C_VEL
LIN {X 0,Y 580.262,Z 197.208,A -85,B 0,C 180,E1 -1691.647,E2 -1691.647} C_VEL
LIN {X 0,Y 580.274,Z 197.203,A -85,B 0,C 180,E1 -1693.827,E2 -1693.827} C_VEL
LIN {X 0,Y 580.32,Z 197.194,A -85,B 0,C 180,E1 -1695.985,E2 -1695.985} C_VEL
LIN {X 0,Y 580.301,Z 197.196,A -85,B 0,C 180,E1 -1698.828,E2 -1698.828} C_VEL
LIN {X 0,Y 580.333,Z 197.196,A -85,B 0,C 180,E1 -1701.645,E2 -1701.645} C_VEL
LIN {X 0,Y 580.321,Z 197.192,A -85,B 0,C 180,E1 -1704.441,E2 -1704.441} C_VEL
LIN {X 0,Y 580.345,Z 197.19,A -85,B 0,C 180,E1 -1707.918,E2 -1707.918} C_VEL
LIN {X 0,Y 580.354,Z 197.19,A -85,B 0,C 180,E1 -1710.694,E2 -1710.694} C_VEL
LIN {X 0,Y 580.289,Z 197.201,A -85,B 0,C 180,E1 -1713.471,E2 -1713.471} C_VEL
LIN {X 0,Y 580.33,Z 197.194,A -85,B 0,C 180,E1 -1715.559,E2 -1715.559} C_VEL
LIN {X 0,Y 580.326,Z 197.192,A -85,B 0,C 180,E1 -1718.355,E2 -1718.355} C_VEL
LIN {X 0,Y 580.297,Z 197.202,A -85,B 0,C 180,E1 -1721.19,E2 -1721.19} C_VEL
LIN {X 0,Y 580.323,Z 197.192,A -85,B 0,C 180,E1 -1724.015,E2 -1724.015} C_VEL
LIN {X 0,Y 580.306,Z 197.204,A -85,B 0,C 180,E1 -1726.912,E2 -1726.912} C_VEL
LIN {X 0,Y 580.299,Z 197.195,A -85,B 0,C 180,E1 -1729.82,E2 -1729.82} C_VEL
LIN {X 0,Y 580.265,Z 197.2,A -85,B 0,C 180,E1 -1732.05,E2 -1732.05} C_VEL
LIN {X 0,Y 580.3,Z 197.199,A -85,B 0,C 180,E1 -1735.077,E2 -1735.077} C_VEL
LIN {X 0,Y 580.307,Z 197.195,A -85,B 0,C 180,E1 -1737.861,E2 -1737.861} C_VEL
LIN {X 0,Y 580.295,Z 197.205,A -85,B 0,C 180,E1 -1740.697,E2 -1740.697} C_VEL
LIN {X 0,Y 580.349,Z 197.341,A -85,B 0,C 180,E1 -1741.733,E2 -1741.733} C_VEL
LIN {X 0,Y 580.368,Z 210.65,A -85,B 0,C 180,E1 -1744.203,E2 -1744.203} C_VEL
LIN {X 0,Y 580.249,Z 222.649,A -85,B 0,C 180,E1 -1746.4,E2 -1746.4} C_VEL
LIN {X 0,Y 580.953,Z 228.393,A -85,B 0,C 180,E1 -1746.491,E2 -1746.491} C_VEL
LIN {X 0,Y 580.758,Z 329.426,A -85,B 0,C 180,E1 -1747.762,E2 -1747.762} C_VEL
LIN {X 0,Y 580.675,Z 342.85,A -85,B 0,C 180,E1 -1748.078,E2 -1748.078} C_VEL
LIN {X 0,Y 580.627,Z 355.198,A -85,B 0,C 180,E1 -1748.513,E2 -1748.513} C_VEL
LIN {X 0,Y 580.548,Z 367.084,A -85,B 0,C 180,E1 -1749.079,E2 -1749.079} C_VEL
LIN {X 0,Y 580.449,Z 377.744,A -85,B 0,C 180,E1 -1749.724,E2 -1749.724} C_VEL
LIN {X 0,Y 580.355,Z 388.364,A -85,B 0,C 180,E1 -1750.527,E2 -1750.527} C_VEL
LIN {X 0,Y 580.285,Z 397.057,A -85,B 0,C 180,E1 -1751.332,E2 -1751.332} C_VEL
LIN {X 0,Y 580.197,Z 406.151,A -85,B 0,C 180,E1 -1752.363,E2 -1752.363} C_VEL
LIN {X 0,Y 580.149,Z 413.375,A -85,B 0,C 180,E1 -1753.378,E2 -1753.378} C_VEL
LIN {X 0,Y 580.122,Z 419.136,A -85,B 0,C 180,E1 -1754.376,E2 -1754.376} C_VEL
LIN {X 0,Y 580.108,Z 424.732,A -85,B 0,C 180,E1 -1755.619,E2 -1755.619} C_VEL
LIN {X 0,Y 580.066,Z 428.117,A -85,B 0,C 180,E1 -1756.625,E2 -1756.625} C_VEL
LIN {X 0,Y 580.062,Z 430.606,A -85,B 0,C 180,E1 -1757.645,E2 -1757.645} C_VEL
LIN {X 0,Y 580.008,Z 432.225,A -85,B 0,C 180,E1 -1758.692,E2 -1758.692} C_VEL
LIN {X 0,Y 580.037,Z 433,A -85,B 0,C 180,E1 -1760.046,E2 -1760.046} C_VEL
LIN {X 0,Y 580.043,Z 432.645,A -85,B 0,C 180,E1 -1760.947,E2 -1760.947} C_VEL
LIN {X 0,Y 580.051,Z 431.484,A -85,B 0,C 180,E1 -1761.949,E2 -1761.949} C_VEL
LIN {X 0,Y 580.058,Z 429.137,A -85,B 0,C 180,E1 -1763.089,E2 -1763.089} C_VEL
LIN {X 0,Y 580.098,Z 424.846,A -85,B 0,C 180,E1 -1764.442,E2 -1764.442} C_VEL
LIN {X 0,Y 580.074,Z 420.4,A -85,B 0,C 180,E1 -1765.465,E2 -1765.465} C_VEL
LIN {X 0,Y 580.138,Z 415.069,A -85,B 0,C 180,E1 -1766.441,E2 -1766.441} C_VEL
LIN {X 0,Y 580.181,Z 407.242,A -85,B 0,C 180,E1 -1767.587,E2 -1767.587} C_VEL
LIN {X 0,Y 580.266,Z 398.454,A -85,B 0,C 180,E1 -1768.614,E2 -1768.614} C_VEL
LIN {X 0,Y 580.362,Z 388.751,A -85,B 0,C 180,E1 -1769.53,E2 -1769.53} C_VEL
LIN {X 0,Y 580.405,Z 377.903,A -85,B 0,C 180,E1 -1770.355,E2 -1770.355} C_VEL
LIN {X 0,Y 580.53,Z 366.607,A -85,B 0,C 180,E1 -1771.037,E2 -1771.037} C_VEL
LIN {X 0,Y 580.669,Z 354.915,A -85,B 0,C 180,E1 -1771.588,E2 -1771.588} C_VEL
LIN {X 0,Y 580.717,Z 341.892,A -85,B 0,C 180,E1 -1772.039,E2 -1772.039} C_VEL
LIN {X 0,Y 580.789,Z 329.114,A -85,B 0,C 180,E1 -1772.334,E2 -1772.334} C_VEL
LIN {X 0,Y 580.924,Z 226.4,A -85,B 0,C 180,E1 -1773.625,E2 -1773.625} C_VEL
LIN {X 0,Y 580.292,Z 222.576,A -85,B 0,C 180,E1 -1773.702,E2 -1773.702} C_VEL
LIN {X 0,Y 580.362,Z 207.623,A -85,B 0,C 180,E1 -1776.446,E2 -1776.446} C_VEL
LIN {X 0,Y 580.281,Z 197.289,A -85,B 0,C 180,E1 -1778.369,E2 -1778.369} C_VEL
LIN {X 0,Y 580.282,Z 197.2,A -85,B 0,C 180,E1 -1780.913,E2 -1780.913} C_VEL
LIN {X 0,Y 580.249,Z 197.205,A -85,B 0,C 180,E1 -1783.825,E2 -1783.825} C_VEL
LIN {X 0,Y 580.251,Z 197.203,A -85,B 0,C 180,E1 -1786.696,E2 -1786.696} C_VEL
LIN {X 0,Y 580.274,Z 197.205,A -85,B 0,C 180,E1 -1789.533,E2 -1789.533} C_VEL
LIN {X 0,Y 580.285,Z 197.197,A -85,B 0,C 180,E1 -1792.344,E2 -1792.344} C_VEL
LIN {X 0,Y 580.299,Z 197.205,A -85,B 0,C 180,E1 -1795.137,E2 -1795.137} C_VEL
LIN {X 0,Y 580.276,Z 197.198,A -85,B 0,C 180,E1 -1797.918,E2 -1797.918} C_VEL
LIN {X 0,Y 580.319,Z 197.197,A -85,B 0,C 180,E1 -1800.694,E2 -1800.694} C_VEL
LIN {X 0,Y 580.245,Z 197.205,A -85,B 0,C 180,E1 -1803.472,E2 -1803.472} C_VEL
LIN {X 0,Y 580.275,Z 197.199,A -85,B 0,C 180,E1 -1805.56,E2 -1805.56} C_VEL
LIN {X 0,Y 580.276,Z 197.2,A -85,B 0,C 180,E1 -1808.357,E2 -1808.357} C_VEL
LIN {X 0,Y 580.325,Z 197.195,A -85,B 0,C 180,E1 -1811.234,E2 -1811.234} C_VEL
LIN {X 0,Y 580.258,Z 197.203,A -85,B 0,C 180,E1 -1814.34,E2 -1814.34} C_VEL
LIN {X 0,Y 580.29,Z 197.203,A -85,B 0,C 180,E1 -1816.927,E2 -1816.927} C_VEL
LIN {X 0,Y 580.262,Z 197.199,A -85,B 0,C 180,E1 -1819.824,E2 -1819.824} C_VEL
LIN {X 0,Y 580.279,Z 197.204,A -85,B 0,C 180,E1 -1822.803,E2 -1822.803} C_VEL
LIN {X 0,Y 580.257,Z 197.203,A -85,B 0,C 180,E1 -1825.082,E2 -1825.082} C_VEL
LIN {X 0,Y 580.277,Z 197.199,A -85,B 0,C 180,E1 -1827.866,E2 -1827.866} C_VEL
LIN {X 0,Y 580.249,Z 197.208,A -85,B 0,C 180,E1 -1830.699,E2 -1830.699} C_VEL
LIN {X 0,Y 580.261,Z 197.2,A -85,B 0,C 180,E1 -1833.319,E2 -1833.319} C_VEL
LIN {X 0,Y 580.288,Z 197.197,A -85,B 0,C 180,E1 -1835.771,E2 -1835.771} C_VEL
LIN {X 0,Y 580.253,Z 197.207,A -85,B 0,C 180,E1 -1838.149,E2 -1838.149} C_VEL
LIN {X 0,Y 580.267,Z 197.201,A -85,B 0,C 180,E1 -1840.846,E2 -1840.846} C_VEL
LIN {X 0,Y 580.251,Z 197.202,A -85,B 0,C 180,E1 -1843.661,E2 -1843.661} C_VEL
LIN {X 0,Y 580.253,Z 197.204,A -85,B 0,C 180,E1 -1846.612,E2 -1846.612} C_VEL
LIN {X 0,Y 580.275,Z 197.198,A -85,B 0,C 180,E1 -1849.16,E2 -1849.16} C_VEL
LIN {X 0,Y 580.268,Z 197.207,A -85,B 0,C 180,E1 -1851.93,E2 -1851.93} C_VEL
LIN {X 0,Y 580.268,Z 197.202,A -85,B 0,C 180,E1 -1854.458,E2 -1854.458} C_VEL
LIN {X 0,Y 580.274,Z 197.198,A -85,B 0,C 180,E1 -1856.978,E2 -1856.978} C_VEL
LIN {X 0,Y 580.288,Z 197.199,A -85,B 0,C 180,E1 -1859.428,E2 -1859.428} C_VEL
LIN {X 0,Y 580.287,Z 197.203,A -85,B 0,C 180,E1 -1862.144,E2 -1862.144} C_VEL
LIN {X 0,Y 580.314,Z 197.196,A -85,B 0,C 180,E1 -1865.272,E2 -1865.272} C_VEL
LIN {X 0,Y 580.3,Z 197.228,A -85,B 0,C 180,E1 -1866.304,E2 -1866.304} C_VEL
LIN {X 0,Y 580.928,Z 201.839,A -85,B 0,C 180,E1 -1866.955,E2 -1866.955} C_VEL
LIN {X 0,Y 580.848,Z 220.096,A -85,B 0,C 180,E1 -1869.461,E2 -1869.461} C_VEL
LIN {X 0,Y 580.61,Z 241.368,A -85,B 0,C 180,E1 -1872.387,E2 -1872.387} C_VEL
LIN {X 0,Y 580.455,Z 261.31,A -85,B 0,C 180,E1 -1875.092,E2 -1875.092} C_VEL
LIN {X 0,Y 580.412,Z 270.533,A -85,B 0,C 180,E1 -1876.333,E2 -1876.333} C_VEL
LIN {X 0,Y 580.958,Z 276.627,A -85,B 0,C 180,E1 -1876.424,E2 -1876.424} C_VEL
LIN {X 0,Y 580.771,Z 379.015,A -85,B 0,C 180,E1 -1877.709,E2 -1877.709} C_VEL
LIN {X 0,Y 580.696,Z 392.263,A -85,B 0,C 180,E1 -1878.017,E2 -1878.017} C_VEL
LIN {X 0,Y 580.652,Z 405.169,A -85,B 0,C 180,E1 -1878.467,E2 -1878.467} C_VEL
LIN {X 0,Y 580.552,Z 416.649,A -85,B 0,C 180,E1 -1879.01,E2 -1879.01} C_VEL
LIN {X 0,Y 580.444,Z 428.218,A -85,B 0,C 180,E1 -1879.713,E2 -1879.713} C_VEL
LIN {X 0,Y 580.344,Z 438.612,A -85,B 0,C 180,E1 -1880.504,E2 -1880.504} C_VEL
LIN {X 0,Y 580.271,Z 447.122,A -85,B 0,C 180,E1 -1881.293,E2 -1881.293} C_VEL
LIN {X 0,Y 580.221,Z 454.967,A -85,B 0,C 180,E1 -1882.169,E2 -1882.169} C_VEL
LIN {X 0,Y 580.153,Z 462.655,A -85,B 0,C 180,E1 -1883.222,E2 -1883.222} C_VEL
LIN {X 0,Y 580.139,Z 469.683,A -85,B 0,C 180,E1 -1884.439,E2 -1884.439} C_VEL
LIN {X 0,Y 580.108,Z 474.374,A -85,B 0,C 180,E1 -1885.484,E2 -1885.484} C_VEL
LIN {X 0,Y 580.123,Z 477.958,A -85,B 0,C 180,E1 -1886.528,E2 -1886.528} C_VEL
LIN {X 0,Y 580.043,Z 479.809,A -85,B 0,C 180,E1 -1887.222,E2 -1887.222} C_VEL
LIN {X 0,Y 580.04,Z 481.199,A -85,B 0,C 180,E1 -1887.917,E2 -1887.917} C_VEL
LIN {X 0,Y 580.04,Z 482.785,A -85,B 0,C 180,E1 -1889.306,E2 -1889.306} C_VEL
LIN {X 0,Y 580.037,Z 483,A -85,B 0,C 180,E1 -1890,E2 -1890} C_VEL
LIN {X 0,Y 580.046,Z 482.186,A -85,B 0,C 180,E1 -1891.388,E2 -1891.388} C_VEL
LIN {X 0,Y 580.04,Z 481.2,A -85,B 0,C 180,E1 -1892.083,E2 -1892.083} C_VEL
LIN {X 0,Y 580.043,Z 479.811,A -85,B 0,C 180,E1 -1892.778,E2 -1892.778} C_VEL
LIN {X 0,Y 580.11,Z 476.897,A -85,B 0,C 180,E1 -1893.82,E2 -1893.82} C_VEL
LIN {X 0,Y 580.053,Z 472.951,A -85,B 0,C 180,E1 -1894.865,E2 -1894.865} C_VEL
LIN {X 0,Y 580.139,Z 466.881,A -85,B 0,C 180,E1 -1896.084,E2 -1896.084} C_VEL
LIN {X 0,Y 580.184,Z 460.244,A -85,B 0,C 180,E1 -1897.132,E2 -1897.132} C_VEL
LIN {X 0,Y 580.25,Z 451.999,A -85,B 0,C 180,E1 -1898.181,E2 -1898.181} C_VEL
LIN {X 0,Y 580.307,Z 443.55,A -85,B 0,C 180,E1 -1899.057,E2 -1899.057} C_VEL
LIN {X 0,Y 580.425,Z 433.113,A -85,B 0,C 180,E1 -1899.935,E2 -1899.935} C_VEL
LIN {X 0,Y 580.492,Z 422.775,A -85,B 0,C 180,E1 -1900.638,E2 -1900.638} C_VEL
LIN {X 0,Y 580.594,Z 411.27,A -85,B 0,C 180,E1 -1901.263,E2 -1901.263} C_VEL
LIN {X 0,Y 580.677,Z 398.512,A -85,B 0,C 180,E1 -1901.784,E2 -1901.784} C_VEL
LIN {X 0,Y 580.781,Z 385.493,A -85,B 0,C 180,E1 -1902.158,E2 -1902.158} C_VEL
LIN {X 0,Y 580.81,Z 373.19,A -85,B 0,C 180,E1 -1902.379,E2 -1902.379} C_VEL
LIN {X 0,Y 580.811,Z 273.285,A -85,B 0,C 180,E1 -1903.621,E2 -1903.621} C_VEL
LIN {X 0,Y 580.418,Z 270.451,A -85,B 0,C 180,E1 -1903.678,E2 -1903.678} C_VEL
LIN {X 0,Y 580.595,Z 248.016,A -85,B 0,C 180,E1 -1906.706,E2 -1906.706} C_VEL
LIN {X 0,Y 580.777,Z 226.604,A -85,B 0,C 180,E1 -1909.639,E2 -1909.639} C_VEL
LIN {X 0,Y 580.943,Z 206.676,A -85,B 0,C 180,E1 -1912.397,E2 -1912.397} C_VEL
LIN {X 0,Y 580.86,Z 200.266,A -85,B 0,C 180,E1 -1913.289,E2 -1913.289} C_VEL
LIN {X 0,Y 580.276,Z 197.206,A -85,B 0,C 180,E1 -1913.745,E2 -1913.745} C_VEL
LIN {X 0,Y 580.281,Z 197.205,A -85,B 0,C 180,E1 -1916.331,E2 -1916.331} C_VEL
LIN {X 0,Y 580.289,Z 197.197,A -85,B 0,C 180,E1 -1919.307,E2 -1919.307} C_VEL
LIN {X 0,Y 580.281,Z 197.204,A -85,B 0,C 180,E1 -1922.198,E2 -1922.198} C_VEL
LIN {X 0,Y 580.271,Z 197.199,A -85,B 0,C 180,E1 -1924.693,E2 -1924.693} C_VEL
LIN {X 0,Y 580.278,Z 197.198,A -85,B 0,C 180,E1 -1927.265,E2 -1927.265} C_VEL
LIN {X 0,Y 580.273,Z 197.202,A -85,B 0,C 180,E1 -1930.268,E2 -1930.268} C_VEL
LIN {X 0,Y 580.252,Z 197.201,A -85,B 0,C 180,E1 -1932.703,E2 -1932.703} C_VEL
LIN {X 0,Y 580.238,Z 197.209,A -85,B 0,C 180,E1 -1935.606,E2 -1935.606} C_VEL
LIN {X 0,Y 580.28,Z 197.2,A -85,B 0,C 180,E1 -1938.231,E2 -1938.231} C_VEL
LIN {X 0,Y 580.244,Z 197.202,A -85,B 0,C 180,E1 -1940.962,E2 -1940.962} C_VEL
LIN {X 0,Y 580.259,Z 197.21,A -85,B 0,C 180,E1 -1943.595,E2 -1943.595} C_VEL
LIN {X 0,Y 580.281,Z 197.199,A -85,B 0,C 180,E1 -1946.143,E2 -1946.143} C_VEL
LIN {X 0,Y 580.248,Z 197.201,A -85,B 0,C 180,E1 -1948.613,E2 -1948.613} C_VEL
LIN {X 0,Y 580.26,Z 197.203,A -85,B 0,C 180,E1 -1951.022,E2 -1951.022} C_VEL
LIN {X 0,Y 580.279,Z 197.204,A -85,B 0,C 180,E1 -1953.656,E2 -1953.656} C_VEL
LIN {X 0,Y 580.252,Z 197.2,A -85,B 0,C 180,E1 -1956.441,E2 -1956.441} C_VEL
LIN {X 0,Y 580.246,Z 197.21,A -85,B 0,C 180,E1 -1959.436,E2 -1959.436} C_VEL
LIN {X 0,Y 580.24,Z 197.206,A -85,B 0,C 180,E1 -1961.644,E2 -1961.644} C_VEL
LIN {X 0,Y 580.239,Z 197.204,A -85,B 0,C 180,E1 -1963.824,E2 -1963.824} C_VEL
LIN {X 0,Y 580.229,Z 197.206,A -85,B 0,C 180,E1 -1966.695,E2 -1966.695} C_VEL
LIN {X 0,Y 580.331,Z 197.195,A -85,B 0,C 180,E1 -1968.827,E2 -1968.827} C_VEL
LIN {X 0,Y 580.276,Z 197.2,A -85,B 0,C 180,E1 -1971.643,E2 -1971.643} C_VEL
LIN {X 0,Y 580.274,Z 197.199,A -85,B 0,C 180,E1 -1974.44,E2 -1974.44} C_VEL
LIN {X 0,Y 580.296,Z 197.201,A -85,B 0,C 180,E1 -1977.223,E2 -1977.223} C_VEL
LIN {X 0,Y 580.285,Z 197.196,A -85,B 0,C 180,E1 -1980,E2 -1980} C_VEL
LIN {X 0,Y 580.302,Z 197.203,A -85,B 0,C 180,E1 -1982.776,E2 -1982.776} C_VEL
LIN {X 0,Y 580.278,Z 197.198,A -85,B 0,C 180,E1 -1985.56,E2 -1985.56} C_VEL
LIN {X 0,Y 580.284,Z 197.197,A -85,B 0,C 180,E1 -1987.656,E2 -1987.656} C_VEL
LIN {X 0,Y 580.272,Z 197.204,A -85,B 0,C 180,E1 -1990.467,E2 -1990.467} C_VEL
LIN {X 0,Y 580.25,Z 197.202,A -85,B 0,C 180,E1 -1993.304,E2 -1993.304} C_VEL
LIN {X 0,Y 580.247,Z 197.204,A -85,B 0,C 180,E1 -1996.175,E2 -1996.175} C_VEL
LIN {X 0,Y 580.271,Z 197.2,A -85,B 0,C 180,E1 -1999.162,E2 -1999.162} C_VEL
LIN {X 0,Y 580.272,Z 197.198,A -85,B 0,C 180,E1 -2001.375,E2 -2001.375} C_VEL
LIN {X 0,Y 579.59,Z 197.286,A -85,B 0,C 180,E1 -2001.955,E2 -2001.955} C_VEL
LIN {X 0,Y 576.715,Z 197.645,A -85,B 0,C 180,E1 -2002.895,E2 -2002.895} C_VEL
LIN {X 0,Y 574.305,Z 197.943,A -85,B 0,C 180,E1 -2003.651,E2 -2003.651} C_VEL
LIN {X 0,Y 573.288,Z 198.074,A -85,B 0,C 180,E1 -2004.235,E2 -2004.235} C_VEL
LIN {X 0,Y 573.214,Z 198.082,A -85,B 0,C 180,E1 -2004.433,E2 -2004.433} C_VEL
LIN {X 0,Y 573.224,Z 198.078,A -85,B 0,C 180,E1 -2006.977,E2 -2006.977} C_VEL
LIN {X 0,Y 573.221,Z 198.077,A -85,B 0,C 180,E1 -2009.495,E2 -2009.495} C_VEL
LIN {X 0,Y 573.22,Z 198.081,A -85,B 0,C 180,E1 -2012.647,E2 -2012.647} C_VEL
LIN {X 0,Y 573.229,Z 198.075,A -85,B 0,C 180,E1 -2015.186,E2 -2015.186} C_VEL
LIN {X 0,Y 573.201,Z 198.083,A -85,B 0,C 180,E1 -2017.81,E2 -2017.81} C_VEL
LIN {X 0,Y 573.264,Z 198.075,A -85,B 0,C 180,E1 -2020.535,E2 -2020.535} C_VEL
LIN {X 0,Y 573.222,Z 198.08,A -85,B 0,C 180,E1 -2023.673,E2 -2023.673} C_VEL
LIN {X 0,Y 573.216,Z 198.079,A -85,B 0,C 180,E1 -2026.645,E2 -2026.645} C_VEL
LIN {X 0,Y 573.246,Z 198.076,A -85,B 0,C 180,E1 -2029.481,E2 -2029.481} C_VEL
LIN {X 0,Y 573.214,Z 198.083,A -85,B 0,C 180,E1 -2032.196,E2 -2032.196} C_VEL
LIN {X 0,Y 573.247,Z 198.073,A -85,B 0,C 180,E1 -2034.82,E2 -2034.82} C_VEL
LIN {X 0,Y 573.238,Z 198.077,A -85,B 0,C 180,E1 -2037.358,E2 -2037.358} C_VEL
LIN {X 0,Y 573.24,Z 198.084,A -85,B 0,C 180,E1 -2039.827,E2 -2039.827} C_VEL
LIN {X 0,Y 573.274,Z 198.072,A -85,B 0,C 180,E1 -2042.238,E2 -2042.238} C_VEL
LIN {X 0,Y 573.258,Z 198.074,A -85,B 0,C 180,E1 -2045.124,E2 -2045.124} C_VEL
LIN {X 0,Y 573.227,Z 198.085,A -85,B 0,C 180,E1 -2047.664,E2 -2047.664} C_VEL
LIN {X 0,Y 573.27,Z 198.07,A -85,B 0,C 180,E1 -2050.73,E2 -2050.73} C_VEL
LIN {X 0,Y 573.246,Z 198.082,A -85,B 0,C 180,E1 -2053.624,E2 -2053.624} C_VEL
LIN {X 0,Y 573.268,Z 198.075,A -85,B 0,C 180,E1 -2055.809,E2 -2055.809} C_VEL
LIN {X 0,Y 573.26,Z 198.073,A -85,B 0,C 180,E1 -2058.746,E2 -2058.746} C_VEL
LIN {X 0,Y 573.288,Z 198.075,A -85,B 0,C 180,E1 -2061.542,E2 -2061.542} C_VEL
LIN {X 0,Y 573.29,Z 198.068,A -85,B 0,C 180,E1 -2064.373,E2 -2064.373} C_VEL
LIN {X 0,Y 573.315,Z 198.066,A -85,B 0,C 180,E1 -2067.893,E2 -2067.893} C_VEL
LIN {X 0,Y 573.325,Z 198.066,A -85,B 0,C 180,E1 -2070.702,E2 -2070.702} C_VEL
LIN {X 0,Y 573.299,Z 198.071,A -85,B 0,C 180,E1 -2072.81,E2 -2072.81} C_VEL
LIN {X 0,Y 573.296,Z 198.069,A -85,B 0,C 180,E1 -2075.628,E2 -2075.628} C_VEL
LIN {X 0,Y 573.282,Z 198.071,A -85,B 0,C 180,E1 -2078.459,E2 -2078.459} C_VEL
LIN {X 0,Y 573.269,Z 198.075,A -85,B 0,C 180,E1 -2081.311,E2 -2081.311} C_VEL
LIN {X 0,Y 573.277,Z 198.072,A -85,B 0,C 180,E1 -2084.423,E2 -2084.423} C_VEL
LIN {X 0,Y 573.254,Z 198.078,A -85,B 0,C 180,E1 -2087.11,E2 -2087.11} C_VEL
LIN {X 0,Y 573.249,Z 198.074,A -85,B 0,C 180,E1 -2090.074,E2 -2090.074} C_VEL
LIN {X 0,Y 573.229,Z 198.079,A -85,B 0,C 180,E1 -2092.336,E2 -2092.336} C_VEL
LIN {X 0,Y 573.249,Z 198.075,A -85,B 0,C 180,E1 -2095.407,E2 -2095.407} C_VEL
LIN {X 0,Y 573.252,Z 198.075,A -85,B 0,C 180,E1 -2098.029,E2 -2098.029} C_VEL
LIN {X 0,Y 573.257,Z 198.081,A -85,B 0,C 180,E1 -2100.887,E2 -2100.887} C_VEL
LIN {X 0,Y 573.309,Z 198.142,A -85,B 0,C 180,E1 -2101.653,E2 -2101.653} C_VEL
LIN {X 0,Y 573.38,Z 208.175,A -85,B 0,C 180,E1 -2103.542,E2 -2103.542} C_VEL
LIN {X 0,Y 573.214,Z 222.617,A -85,B 0,C 180,E1 -2106.224,E2 -2106.224} C_VEL
LIN {X 0,Y 574.028,Z 227.567,A -85,B 0,C 180,E1 -2106.314,E2 -2106.314} C_VEL
LIN {X 0,Y 573.834,Z 329.413,A -85,B 0,C 180,E1 -2107.611,E2 -2107.611} C_VEL
LIN {X 0,Y 573.717,Z 342.461,A -85,B 0,C 180,E1 -2107.919,E2 -2107.919} C_VEL
LIN {X 0,Y 573.683,Z 355.124,A -85,B 0,C 180,E1 -2108.368,E2 -2108.368} C_VEL
LIN {X 0,Y 573.571,Z 367.223,A -85,B 0,C 180,E1 -2108.952,E2 -2108.952} C_VEL
LIN {X 0,Y 573.438,Z 377.584,A -85,B 0,C 180,E1 -2109.586,E2 -2109.586} C_VEL
LIN {X 0,Y 573.368,Z 388.175,A -85,B 0,C 180,E1 -2110.394,E2 -2110.394} C_VEL
LIN {X 0,Y 573.22,Z 398.12,A -85,B 0,C 180,E1 -2111.335,E2 -2111.335} C_VEL
LIN {X 0,Y 573.118,Z 407.218,A -85,B 0,C 180,E1 -2112.406,E2 -2112.406} C_VEL
LIN {X 0,Y 573.064,Z 413.85,A -85,B 0,C 180,E1 -2113.37,E2 -2113.37} C_VEL
LIN {X 0,Y 573.03,Z 419.35,A -85,B 0,C 180,E1 -2114.347,E2 -2114.347} C_VEL
LIN {X 0,Y 573.023,Z 423.844,A -85,B 0,C 180,E1 -2115.339,E2 -2115.339} C_VEL
LIN {X 0,Y 572.968,Z 428.213,A -85,B 0,C 180,E1 -2116.616,E2 -2116.616} C_VEL
LIN {X 0,Y 572.987,Z 430.527,A -85,B 0,C 180,E1 -2117.577,E2 -2117.577} C_VEL
LIN {X 0,Y 572.926,Z 432.049,A -85,B 0,C 180,E1 -2118.516,E2 -2118.516} C_VEL
LIN {X 0,Y 572.956,Z 432.881,A -85,B 0,C 180,E1 -2119.501,E2 -2119.501} C_VEL
LIN {X 0,Y 572.924,Z 432.876,A -85,B 0,C 180,E1 -2120.6,E2 -2120.6} C_VEL
LIN {X 0,Y 572.952,Z 431.879,A -85,B 0,C 180,E1 -2121.717,E2 -2121.717} C_VEL
LIN {X 0,Y 572.975,Z 429.311,A -85,B 0,C 180,E1 -2123.057,E2 -2123.057} C_VEL
LIN {X 0,Y 573.022,Z 425.128,A -85,B 0,C 180,E1 -2124.423,E2 -2124.423} C_VEL
LIN {X 0,Y 572.993,Z 419.798,A -85,B 0,C 180,E1 -2125.653,E2 -2125.653} C_VEL
LIN {X 0,Y 573.074,Z 413.878,A -85,B 0,C 180,E1 -2126.716,E2 -2126.716} C_VEL
LIN {X 0,Y 573.132,Z 406.476,A -85,B 0,C 180,E1 -2127.781,E2 -2127.781} C_VEL
LIN {X 0,Y 573.244,Z 397.655,A -85,B 0,C 180,E1 -2128.803,E2 -2128.803} C_VEL
LIN {X 0,Y 573.334,Z 387.808,A -85,B 0,C 180,E1 -2129.728,E2 -2129.728} C_VEL
LIN {X 0,Y 573.415,Z 376.982,A -85,B 0,C 180,E1 -2130.544,E2 -2130.544} C_VEL
LIN {X 0,Y 573.561,Z 365.116,A -85,B 0,C 180,E1 -2131.253,E2 -2131.253} C_VEL
LIN {X 0,Y 573.701,Z 353.178,A -85,B 0,C 180,E1 -2131.8,E2 -2131.8} C_VEL
LIN {X 0,Y 573.784,Z 339.786,A -85,B 0,C 180,E1 -2132.246,E2 -2132.246} C_VEL
LIN {X 0,Y 573.875,Z 326.589,A -85,B 0,C 180,E1 -2132.526,E2 -2132.526} C_VEL
LIN {X 0,Y 573.97,Z 226.96,A -85,B 0,C 180,E1 -2133.785,E2 -2133.785} C_VEL
LIN {X 0,Y 573.254,Z 222.652,A -85,B 0,C 180,E1 -2133.859,E2 -2133.859} C_VEL
LIN {X 0,Y 573.331,Z 208.326,A -85,B 0,C 180,E1 -2136.521,E2 -2136.521} C_VEL
LIN {X 0,Y 573.381,Z 200.197,A -85,B 0,C 180,E1 -2138.048,E2 -2138.048} C_VEL
LIN {X 0,Y 573.248,Z 198.077,A -85,B 0,C 180,E1 -2138.47,E2 -2138.47} C_VEL
LIN {X 0,Y 573.207,Z 198.088,A -85,B 0,C 180,E1 -2141.411,E2 -2141.411} C_VEL
LIN {X 0,Y 573.223,Z 198.084,A -85,B 0,C 180,E1 -2143.621,E2 -2143.621} C_VEL
LIN {X 0,Y 573.205,Z 198.08,A -85,B 0,C 180,E1 -2146.529,E2 -2146.529} C_VEL
LIN {X 0,Y 573.248,Z 198.082,A -85,B 0,C 180,E1 -2149.403,E2 -2149.403} C_VEL
LIN {X 0,Y 573.235,Z 198.075,A -85,B 0,C 180,E1 -2152.25,E2 -2152.25} C_VEL
LIN {X 0,Y 573.245,Z 198.074,A -85,B 0,C 180,E1 -2154.372,E2 -2154.372} C_VEL
LIN {X 0,Y 573.267,Z 198.08,A -85,B 0,C 180,E1 -2157.189,E2 -2157.189} C_VEL
LIN {X 0,Y 573.256,Z 198.073,A -85,B 0,C 180,E1 -2160,E2 -2160} C_VEL
LIN {X 0,Y 573.262,Z 198.078,A -85,B 0,C 180,E1 -2162.811,E2 -2162.811} C_VEL
LIN {X 0,Y 573.239,Z 198.075,A -85,B 0,C 180,E1 -2165.629,E2 -2165.629} C_VEL
LIN {X 0,Y 573.249,Z 198.076,A -85,B 0,C 180,E1 -2168.46,E2 -2168.46} C_VEL
LIN {X 0,Y 573.269,Z 198.073,A -85,B 0,C 180,E1 -2171.312,E2 -2171.312} C_VEL
LIN {X 0,Y 573.224,Z 198.08,A -85,B 0,C 180,E1 -2174.426,E2 -2174.426} C_VEL
LIN {X 0,Y 573.248,Z 198.077,A -85,B 0,C 180,E1 -2177.112,E2 -2177.112} C_VEL
LIN {X 0,Y 573.213,Z 198.079,A -85,B 0,C 180,E1 -2180.078,E2 -2180.078} C_VEL
LIN {X 0,Y 573.222,Z 198.078,A -85,B 0,C 180,E1 -2183.156,E2 -2183.156} C_VEL
LIN {X 0,Y 573.24,Z 198.078,A -85,B 0,C 180,E1 -2186.191,E2 -2186.191} C_VEL
LIN {X 0,Y 573.204,Z 198.088,A -85,B 0,C 180,E1 -2188.567,E2 -2188.567} C_VEL
LIN {X 0,Y 573.194,Z 198.082,A -85,B 0,C 180,E1 -2190.996,E2 -2190.996} C_VEL
LIN {X 0,Y 573.221,Z 198.077,A -85,B 0,C 180,E1 -2193.527,E2 -2193.527} C_VEL
LIN {X 0,Y 573.223,Z 198.08,A -85,B 0,C 180,E1 -2196.051,E2 -2196.051} C_VEL
LIN {X 0,Y 573.208,Z 198.083,A -85,B 0,C 180,E1 -2198.705,E2 -2198.705} C_VEL
LIN {X 0,Y 573.206,Z 198.079,A -85,B 0,C 180,E1 -2201.459,E2 -2201.459} C_VEL
LIN {X 0,Y 573.205,Z 198.087,A -85,B 0,C 180,E1 -2204.337,E2 -2204.337} C_VEL
LIN {X 0,Y 573.215,Z 198.078,A -85,B 0,C 180,E1 -2207.362,E2 -2207.362} C_VEL
LIN {X 0,Y 573.224,Z 198.082,A -85,B 0,C 180,E1 -2210.396,E2 -2210.396} C_VEL
LIN {X 0,Y 573.235,Z 198.075,A -85,B 0,C 180,E1 -2213.081,E2 -2213.081} C_VEL
LIN {X 0,Y 573.25,Z 198.078,A -85,B 0,C 180,E1 -2215.674,E2 -2215.674} C_VEL
LIN {X 0,Y 573.225,Z 198.083,A -85,B 0,C 180,E1 -2218.187,E2 -2218.187} C_VEL
LIN {X 0,Y 573.253,Z 198.075,A -85,B 0,C 180,E1 -2220.637,E2 -2220.637} C_VEL
LIN {X 0,Y 573.209,Z 198.08,A -85,B 0,C 180,E1 -2223.025,E2 -2223.025} C_VEL
LIN {X 0,Y 573.267,Z 198.075,A -85,B 0,C 180,E1 -2225.369,E2 -2225.369} C_VEL
LIN {X 0,Y 573.264,Z 198.217,A -85,B 0,C 180,E1 -2226.204,E2 -2226.204} C_VEL
LIN {X 0,Y 573.956,Z 203.32,A -85,B 0,C 180,E1 -2226.934,E2 -2226.934} C_VEL
LIN {X 0,Y 573.876,Z 222.59,A -85,B 0,C 180,E1 -2229.575,E2 -2229.575} C_VEL
LIN {X 0,Y 573.604,Z 244.292,A -85,B 0,C 180,E1 -2232.57,E2 -2232.57} C_VEL
LIN {X 0,Y 573.465,Z 263.789,A -85,B 0,C 180,E1 -2235.245,E2 -2235.245} C_VEL
LIN {X 0,Y 573.415,Z 270.533,A -85,B 0,C 180,E1 -2236.163,E2 -2236.163} C_VEL
LIN {X 0,Y 574.061,Z 276.627,A -85,B 0,C 180,E1 -2236.258,E2 -2236.258} C_VEL
LIN {X 0,Y 573.833,Z 379.014,A -85,B 0,C 180,E1 -2237.558,E2 -2237.558} C_VEL
LIN {X 0,Y 573.766,Z 392.263,A -85,B 0,C 180,E1 -2237.87,E2 -2237.87} C_VEL
LIN {X 0,Y 573.661,Z 404.407,A -85,B 0,C 180,E1 -2238.294,E2 -2238.294} C_VEL
LIN {X 0,Y 573.579,Z 416.647,A -85,B 0,C 180,E1 -2238.874,E2 -2238.874} C_VEL
LIN {X 0,Y 573.435,Z 428.215,A -85,B 0,C 180,E1 -2239.586,E2 -2239.586} C_VEL
LIN {X 0,Y 573.332,Z 438.614,A -85,B 0,C 180,E1 -2240.387,E2 -2240.387} C_VEL
LIN {X 0,Y 573.24,Z 447.122,A -85,B 0,C 180,E1 -2241.186,E2 -2241.186} C_VEL
LIN {X 0,Y 573.16,Z 454.967,A -85,B 0,C 180,E1 -2242.072,E2 -2242.072} C_VEL
LIN {X 0,Y 573.073,Z 462.585,A -85,B 0,C 180,E1 -2243.127,E2 -2243.127} C_VEL
LIN {X 0,Y 573.07,Z 469.683,A -85,B 0,C 180,E1 -2244.37,E2 -2244.37} C_VEL
LIN {X 0,Y 573.028,Z 474.374,A -85,B 0,C 180,E1 -2245.428,E2 -2245.428} C_VEL
LIN {X 0,Y 573.022,Z 477.958,A -85,B 0,C 180,E1 -2246.485,E2 -2246.485} C_VEL
LIN {X 0,Y 572.959,Z 479.809,A -85,B 0,C 180,E1 -2247.188,E2 -2247.188} C_VEL
LIN {X 0,Y 572.946,Z 482.185,A -85,B 0,C 180,E1 -2248.594,E2 -2248.594} C_VEL
LIN {X 0,Y 572.938,Z 483,A -85,B 0,C 180,E1 -2250,E2 -2250} C_VEL
LIN {X 0,Y 572.946,Z 482.186,A -85,B 0,C 180,E1 -2251.406,E2 -2251.406} C_VEL
LIN {X 0,Y 572.939,Z 481.199,A -85,B 0,C 180,E1 -2252.109,E2 -2252.109} C_VEL
LIN {X 0,Y 572.959,Z 479.811,A -85,B 0,C 180,E1 -2252.812,E2 -2252.812} C_VEL
LIN {X 0,Y 573.014,Z 476.897,A -85,B 0,C 180,E1 -2253.867,E2 -2253.867} C_VEL
LIN {X 0,Y 572.963,Z 472.951,A -85,B 0,C 180,E1 -2254.925,E2 -2254.925} C_VEL
LIN {X 0,Y 573.092,Z 467.871,A -85,B 0,C 180,E1 -2255.983,E2 -2255.983} C_VEL
LIN {X 0,Y 573.103,Z 461.474,A -85,B 0,C 180,E1 -2257.043,E2 -2257.043} C_VEL
LIN {X 0,Y 573.177,Z 453.486,A -85,B 0,C 180,E1 -2258.105,E2 -2258.105} C_VEL
LIN {X 0,Y 573.253,Z 445.346,A -85,B 0,C 180,E1 -2258.992,E2 -2258.992} C_VEL
LIN {X 0,Y 573.349,Z 435.414,A -85,B 0,C 180,E1 -2259.88,E2 -2259.88} C_VEL
LIN {X 0,Y 573.505,Z 424.207,A -85,B 0,C 180,E1 -2260.68,E2 -2260.68} C_VEL
LIN {X 0,Y 573.626,Z 413.202,A -85,B 0,C 180,E1 -2261.304,E2 -2261.304} C_VEL
LIN {X 0,Y 573.703,Z 401.017,A -85,B 0,C 180,E1 -2261.839,E2 -2261.839} C_VEL
LIN {X 0,Y 573.811,Z 388.234,A -85,B 0,C 180,E1 -2262.241,E2 -2262.241} C_VEL
LIN {X 0,Y 573.891,Z 374.7,A -85,B 0,C 180,E1 -2262.508,E2 -2262.508} C_VEL
LIN {X 0,Y 573.919,Z 274.179,A -85,B 0,C 180,E1 -2263.777,E2 -2263.777} C_VEL
LIN {X 0,Y 573.421,Z 270.451,A -85,B 0,C 180,E1 -2263.848,E2 -2263.848} C_VEL
LIN {X 0,Y 573.618,Z 247.386,A -85,B 0,C 180,E1 -2267.002,E2 -2267.002} C_VEL
LIN {X 0,Y 573.866,Z 225.361,A -85,B 0,C 180,E1 -2270.052,E2 -2270.052} C_VEL
LIN {X 0,Y 574.049,Z 205.045,A -85,B 0,C 180,E1 -2272.872,E2 -2272.872} C_VEL
